(* IEC 61131-3 sources: SmartHomeNew/snapshots/2026-05-07, 56 files *)

(* ---- E_Gateway_Command_Type.dut ---- *)
TYPE E_Gateway_Command_Type :
(
    CMD_NONE := 0,
    CMD_SET_SCENARIO := 1,
    CMD_SET_LIGHT := 2,
    CMD_SET_SOCKET := 3,
    CMD_SET_SECURITY := 4,
    CMD_SET_TEMP := 5,
    CMD_SET_VENT := 6,
    CMD_SET_BLINDS := 7,
    CMD_TELEGRAM_MSG := 8,
    CMD_SYNC_TIME := 9,
    CMD_RESET_ERRORS := 10,
    CMD_SET_CONFIG := 11
) USINT;
END_TYPE

(* ---- E_Outdoor_Mode.dut ---- *)
{attribute 'strict'}
TYPE E_Outdoor_Mode :
(
    OUTDOOR_MODE_AUTO := 0,
    OUTDOOR_MODE_PARTY := 1,
    OUTDOOR_MODE_SECURITY := 2,
    OUTDOOR_MODE_ECONOMY := 3,
    OUTDOOR_MODE_MANUAL := 4
) USINT;
END_TYPE

(* ---- ST_DHW_Status.dut ---- *)
{attribute 'pack_mode' := '1'}
TYPE ST_DHW_Status :
STRUCT
    Temp : REAL;
    Pressure : REAL;
    Heating_Pump_On : BOOL;
    Circ_Pump_On : BOOL;
    Warning : BOOL;
    Error : BOOL;
    Error_ID : WORD;
END_STRUCT
END_TYPE

(* ---- ST_Heating_Runtime_Adaptive_Intelligence.dut ---- *)
TYPE ST_Heating_Runtime_Adaptive_Intelligence :
STRUCT
    // ======================================================
    // Adaptive analytics visibility
    // Passive analytics only.
    // No adaptive authority exists.
    // ======================================================
    Adaptive_Analytics_Visible : BOOL;
    Adaptive_Analytics_Degraded : BOOL;
    Adaptive_Analytics_Attention : BOOL;

    // ======================================================
    // Adaptive supervision observation
    // ======================================================
    Supervision_Confidence_Observation : UINT;
    Confidence_Degradation_Visible : BOOL;

    // ======================================================
    // Adaptive runtime observation
    // ======================================================
    Adaptive_Runtime_Observation : UINT;
    Adaptive_Runtime_Stability_Observation : UINT;

    // ======================================================
    // Adaptive anomaly observation weighting
    // ======================================================
    Runtime_Anomaly_Observation_Weight : UINT;
    Cascade_Anomaly_Observation_Weight : UINT;
    OpenTherm_Anomaly_Observation_Weight : UINT;
    Diagnostics_Anomaly_Observation_Weight : UINT;

    // ======================================================
    // Predictive correlation observation
    // ======================================================
    Predictive_Correlation_Observation : UINT;
    Predictive_Correlation_Visible : BOOL;

    // ======================================================
    // Adaptive integrity observation
    // ======================================================
    Sequencing_Confidence_Observation : UINT;
    Ownership_Confidence_Observation : UINT;
    Synchronization_Confidence_Observation : UINT;

    // ======================================================
    // Adaptive analytics status
    // ======================================================
    Status_Code : UINT;
    Status_Text : STRING(128);
END_STRUCT
END_TYPE

(* ---- ST_Heating_Runtime_Event_Buffer.dut ---- *)
TYPE ST_Heating_Runtime_Event_Buffer :
STRUCT
    // ======================================================
    // Runtime phase events
    // ======================================================
    Events : ARRAY[1..32] OF ST_Heating_Runtime_Phase_Event;

    // ======================================================
    // Runtime buffer state
    // ======================================================
    Write_Index : UINT;
    Read_Index : UINT;
    Event_Count : UINT;
    Overflow : BOOL;

    // ======================================================
    // Runtime integrity
    // ======================================================
    Ordering_Integrity_Valid : BOOL;
    Isolation_Integrity_Valid : BOOL;
    Lifecycle_Integrity_Valid : BOOL;

    // ======================================================
    // Runtime visibility
    // ======================================================
    Diagnostics_Visibility_Valid : BOOL;
    Explainability_Visibility_Valid : BOOL;

    // ======================================================
    // Runtime ownership integrity
    // ======================================================
    OpenTherm_Ownership_Valid : BOOL;
    Cascade_Ownership_Valid : BOOL;
    Safety_Ownership_Valid : BOOL;

    // ======================================================
    // Runtime status
    // ======================================================
    Status_Code : UINT;
    Status_Text : STRING(128);
END_STRUCT
END_TYPE

(* ---- ST_Heating_Runtime_Phase_Event.dut ---- *)
TYPE ST_Heating_Runtime_Phase_Event :
STRUCT
    // ======================================================
    // Runtime phase
    // ======================================================
    Phase : E_Heating_Runtime_Phase;

    // ======================================================
    // Event lifecycle
    // ======================================================
    Event_Active : BOOL;
    Event_Completed : BOOL;
    Event_Failed : BOOL;

    // ======================================================
    // Runtime timing
    // ======================================================
    Start_Time_MS : UDINT;
    End_Time_MS : UDINT;
    Duration_MS : UDINT;

    // ======================================================
    // Runtime integrity
    // ======================================================
    Ordering_Valid : BOOL;
    Isolation_Valid : BOOL;

    // ======================================================
    // Runtime status
    // ======================================================
    Status_Code : UINT;
    Status_Text : STRING(128);

    // ======================================================
    // Diagnostics visibility
    // ======================================================
    Diagnostics_Visible : BOOL;
    Explainability_Visible : BOOL;

    // ======================================================
    // Safety integrity
    // ======================================================
    Safety_Integrity_Valid : BOOL;

    // ======================================================
    // Ownership integrity
    // ======================================================
    OpenTherm_Ownership_Valid : BOOL;
    Cascade_Ownership_Valid : BOOL;
END_STRUCT
END_TYPE

(* ---- ST_Modbus_Response.dut ---- *)
TYPE ST_Modbus_Response :
STRUCT
    Busy : BOOL;
    Done : BOOL;
    Error : BOOL;
    Error_Code : WORD;
    Read_Value : ARRAY[1..32] OF WORD;
    Last_Sequence : UDINT;
    Last_Update_MS : UDINT;
END_STRUCT
END_TYPE

(* ---- ST_OpenTherm_Status.dut ---- *)
TYPE ST_OpenTherm_Status :
STRUCT
    Raw_Heartbeat : UDINT;
    Raw_Ack_Seq : UDINT;
    Raw_Online : BOOL;
    Raw_Error : BOOL;
    Raw_Flame : BOOL;
    Raw_Modulation_x10 : UINT;
    Raw_Boiler_Temp_x10 : INT;
    Raw_Status_Word : WORD;
    Raw_Error_Code : WORD;

    Adapter_Online : BOOL;
    Adapter_Error : BOOL;
    Command_Ack : BOOL;
    Command_Timeout : BOOL;
    Heartbeat_Timeout : BOOL;

    Last_Heartbeat : UDINT;
    Last_Heartbeat_MS : UDINT;

    // Transport freshness telemetry
    Heartbeat_Age_MS : UDINT;
    Command_Age_MS : UDINT;
    Last_Command_Ack_Seq : UDINT;

    Adapter_State : E_OpenTherm_Adapter_State;
    Error_State : E_OpenTherm_Error;
END_STRUCT
END_TYPE

(* ---- ST_Ventilation_Config.dut ---- *)
{attribute 'pack_mode' := '1'}
TYPE ST_Ventilation_Config :
STRUCT
    CO2_Threshold : REAL := 800.0;
    Humidity_Threshold : REAL := 65.0;
    Night_Mode_Start : TOD := TOD#23:00;
    Night_Mode_End : TOD := TOD#07:00;
END_STRUCT
END_TYPE

(* ---- ST_Zone_Adapt_State.dut ---- *)
TYPE ST_Zone_Adapt_State :
STRUCT
    Zone_Weight : REAL;
    Confidence : REAL;
    Activations : UDINT;
    Success_Count : UDINT;
    Failure_Count : UDINT;
    Success_Rate : REAL;
    Avg_Result_Value : REAL;
    Last_Update_MS : UDINT;
END_STRUCT
END_TYPE

(* ---- GVL_BEHAVIOR_ADAPT.gvl ---- *)
VAR_GLOBAL
    // Scenario behavior weights.
    // Scalar fields are the active compile-safe source used by PRG_Scenario_Engine.
    // The structured value is kept as a repository-level model reference, but active code does not depend on direct component access to it.
    G_Behavior_Weight_Comfort : REAL := 1.0;
    G_Behavior_Weight_Night : REAL := 1.0;
    G_Behavior_Weight_Preheat : REAL := 1.0;
    G_Behavior_Weight_VentBoost : REAL := 1.0;
    G_Behavior_Weight_AccessSecure : REAL := 1.0;

    G_Behavior_Weights : ST_Behavior_Weights := (
        W_Comfort := 1.0,
        W_Night := 1.0,
        W_Preheat := 1.0,
        W_VentBoost := 1.0,
        W_AccessSecure := 1.0
    );

    G_Scenario_Stats : ARRAY[0..10] OF ST_Scenario_Stats;
    G_VentBoost_Zone_Adapt : ARRAY[1..GVL_CONSTANTS.C_MAX_ZONES] OF ST_Zone_Adapt_State;

    G_Adapt_Profile : E_Adapt_Profile := ADAPT_PROFILE_BALANCED;

    G_Adapt_Enabled : BOOL := TRUE;
    G_Adapt_Learning_Rate : REAL := 0.05;
    G_Adapt_Update_Threshold : INT := 5;

    G_Adapt_Min_Confidence : REAL := 0.30;
    G_Adapt_Default_Zone_Weight : REAL := 1.0;

    G_Confidence_Learning_Rate : REAL := 0.05;
    G_Decay_Factor : REAL := 0.995;

    G_Prev_Humidity : ARRAY[1..GVL_CONSTANTS.C_MAX_ZONES] OF REAL;
    G_Prev_Valid : ARRAY[1..GVL_CONSTANTS.C_MAX_ZONES] OF BOOL;
END_VAR
// >>> BULK_SYNC_ANCHOR: GVL_BEHAVIOR_ADAPT <<<

(* ---- GVL_CONFIG_BACKUP.gvl ---- *)
{attribute 'qualified_only'}
VAR_GLOBAL
    // Full snapshot of configuration
    G_Backup_FloorHeating_Configs : ARRAY[1..GVL_CONSTANTS.C_MAX_HEATING_CIRCUITS] OF ST_FloorHeating_Circuit_Config;

    G_Backup_Max_Active_Manifolds : INT := 0;
    G_Backup_Max_Thermal_Budget : REAL := 0.0;

    // Integrity flag
    G_Backup_Valid : BOOL := FALSE;
END_VAR

(* ---- GVL_CONSTANTS.gvl ---- *)
{attribute 'qualified_only'}
VAR_GLOBAL CONSTANT
    // Размеры массивов (конфигурация системы)
    C_MAX_ZONES            : INT := 16;
    C_MAX_LIGHTING_ZONES   : INT := 32;
    C_MAX_HEATING_CIRCUITS : INT := 16;
    C_MAX_CLIMATE_ZONES    : INT := 16;
    C_MAX_LIGHT_ZONES      : INT := 32;
    C_MAX_SOCKETS          : INT := 36;
    C_MAX_BLINDS           : INT := 20;
    C_MAX_ALARMS           : INT := 20;
    C_MAX_RULES            : INT := 20;
    C_MAX_MANIFOLDS        : INT := 5;
    C_MAX_BOILERS          : INT := 2;
    C_MAX_SUPPLY_FANS      : INT := 3;
    C_MAX_EXHAUST_FANS     : INT := 5;
    C_MAX_SECURITY_SENSORS : INT := 15;
    C_MAX_FLOOD_SENSORS    : INT := 12;
    C_MAX_DOOR_SENSORS     : INT := 8;
    C_MAX_CO_SENSORS       : INT := 8;
    C_MAX_METHANE_SENSORS  : INT := 2;
    C_PRIMARY_METHANE_SENSOR_INDEX : INT := 1;
    C_PRIMARY_EFFECTIVE_GAS_INDEX : INT := 1;
    C_MAX_VENT_UNITS       : INT := 8;
    C_MAX_SUPPLY_TEMPS     : INT := 2;
    C_MAX_SMOKE_SENSORS    : INT := 6;
    C_MAX_SCENARIOS        : INT := 6;
    C_MAX_OUTDOOR_ZONES    : INT := 4;
    C_MAX_ACCESS_CODES     : INT := 10;
    C_MAX_WET_ZONES        : INT := 4;
    C_MAX_CALIBRATIONS     : INT := 20;
    C_MAX_MODULES          : INT := 10;
    C_MAX_CLEANING_MODES   : INT := 3;
    C_MAX_ALLOWED_IPS      : INT := 5;
    C_MAX_VENT_SUPPLY_MODES: INT := 3;
    C_MAX_SECURITY_PHONES  : INT := 5;
    C_MAX_FLOOD_VALVES     : INT := 3;
    C_MAX_HUMIDITY_SENSORS : INT := 8;
    C_MAX_CO2_SENSORS      : INT := 8;
    C_MAX_CIRCUITS_PER_MANIFOLD : INT := 4;
    C_MAX_TREND_DATA_POINTS: INT := 100;
    C_MAX_HISTORY_RECORDS  : INT := 100;
    C_MAX_DEBUG_LOGS       : INT := 1000;
    C_MAX_GATEWAY_COMMANDS : INT := 10;
    C_MAX_STATE_SNAPSHOTS  : INT := 10;
    C_MAX_BLACKBOX_RECORDS : INT := 100;
    C_MAX_PRESENCE_HISTORY : INT := 1008;
    C_MAX_MODBUS_REGISTERS : INT := 201;
    C_MAX_DEDUPLICATION_HISTORY : INT := 100;
    C_MAX_NVRAM_RECORDS    : INT := 100;
    C_MAX_NVRAM_DATA       : INT := 128;

    C_MAX_WATER_ZONES      : INT := 32;

    C_ANALOG_RAW_MAX       : WORD := 27648;
    C_ANALOG_4MA_RAW       : WORD := 5529;
    C_ANALOG_3_6MA_RAW     : WORD := 4976;
    C_ANALOG_21MA_RAW      : WORD := 29030;
    C_ANALOG_10V_MAX_RAW   : WORD := 30000;

    C_MS_IN_SECOND         : UDINT := 1000;
    C_MS_IN_MINUTE         : UDINT := 60000;
    C_MS_IN_HOUR           : UDINT := 3600000;
    C_MS_IN_DAY            : UDINT := 86400000;

    C_BOILER_CASCADE_MIN_DEMAND : REAL := 25.0;
    C_BOILER_CASCADE_HIGH_DEMAND : REAL := 250.0;
    C_BOILER_SETPOINT_MIN : REAL := 35.0;
    C_BOILER_SETPOINT_MAX : REAL := 55.0;
    C_MIN_HEATING_MANIFOLD_PRESSURE : REAL := 0.8;
END_VAR

(* ---- GVL_GATEWAY.gvl ---- *)
{attribute 'qualified_only'}
VAR_GLOBAL
    G_Gateway_Command : ST_Gateway_Command;
    G_Gateway_Command_Received : BOOL;
    G_Gateway_Send_2FA : BOOL;
    G_Gateway_2FA_Code : STRING(6);
    G_Gateway_Telegram_Msg : STRING(200);
    G_Gateway_Send_Telegram : BOOL;
    G_Gateway_HMI_Status_Message : STRING(200);
    G_Gateway_Ping_OK : BOOL;
    G_Gateway_Data_Ready : BOOL;
    G_Gateway_Modbus_Registers : ARRAY[0..GVL_CONSTANTS.C_MAX_MODBUS_REGISTERS-1] OF WORD;
    // === SHADOW POLICY EXPORT ===
    G_Shadow_Alert_Active : BOOL;
    G_Shadow_Dominant_Channel : STRING(32);
    G_Shadow_Policy_Summary_Text : STRING(160);
    G_Shadow_Recent_Activity_Text : STRING(160);
    G_Shadow_Rate_Summary_Text : STRING(160);
    G_Shadow_Total_Fallback_Count : UDINT;
    G_Shadow_Total_Recovery_Count : UDINT;

END_VAR

(* ---- GVL_Heating_Runtime_Observation.gvl ---- *)
VAR_GLOBAL
    G_Runtime_Observer_Lifecycle_State : E_Runtime_Observer_Lifecycle_State := E_Runtime_Observer_Lifecycle_State.ROS_INACTIVE;
    G_Runtime_Observer_Lifecycle_Code : UINT := 0;
    G_Runtime_Observer_Lifecycle_Text : STRING(128) := 'Heating runtime observer inactive';
    G_Runtime_Observer_Commissioning_Required : BOOL := TRUE;
    G_Runtime_Observer_Commissioning_Active : BOOL := FALSE;
    G_Runtime_Observer_Commissioning_Complete : BOOL := FALSE;
    G_Runtime_Observation : ST_Heating_Runtime_Observation;
    G_Runtime_Observation_Publication_Valid : BOOL := FALSE;
    G_Runtime_Observation_Stabilization_Complete : BOOL := FALSE;
    G_Runtime_Observation_Operational : BOOL := FALSE;
    G_Runtime_Observation_Valid : BOOL := FALSE;
    G_Runtime_Observer_Ready : BOOL := FALSE;
    G_Runtime_Observer_Fault : BOOL := FALSE;
    G_Runtime_Observation_Status_Code : UINT := 0;
    G_Runtime_Observation_Status_Text : STRING(128) := 'Heating runtime observation inactive';
    G_Runtime_Observation_ReadOnly : BOOL := TRUE;
    G_Runtime_Observation_Governance_Locked : BOOL := TRUE;
END_VAR

(* ---- GVL_LIGHTING_OUTPUT.gvl ---- *)
VAR_GLOBAL
    AO_Lighting_Levels : ARRAY[1..GVL_CONSTANTS.C_MAX_LIGHT_ZONES] OF UINT;
    AO_Blinds_Positions : ARRAY[1..GVL_CONSTANTS.C_MAX_BLINDS] OF UINT;
    DO_Sockets : ARRAY[1..GVL_CONSTANTS.C_MAX_SOCKETS] OF BOOL;
END_VAR

(* ---- GVL_STATE.gvl ---- *)
{attribute 'qualified_only'}
VAR_GLOBAL
    G_Floor_Temps : ARRAY[1..GVL_CONSTANTS.C_MAX_HEATING_CIRCUITS] OF REAL;
    G_Room_Temps : ARRAY[1..GVL_CONSTANTS.C_MAX_ZONES] OF REAL;
    G_Last_Valid_Room_Temps : ARRAY[1..GVL_CONSTANTS.C_MAX_ZONES] OF REAL;
    G_Last_Valid_Floor_Temps : ARRAY[1..GVL_CONSTANTS.C_MAX_HEATING_CIRCUITS] OF REAL;
    G_Temp_Sensor_Fault : ARRAY[1..GVL_CONSTANTS.C_MAX_ZONES] OF BOOL;
    G_Floor_Temp_Sensor_Fault : ARRAY[1..GVL_CONSTANTS.C_MAX_HEATING_CIRCUITS] OF BOOL;
    G_Room_Hum : ARRAY[1..GVL_CONSTANTS.C_MAX_ZONES] OF REAL;
    G_Room_CO2 : ARRAY[1..GVL_CONSTANTS.C_MAX_ZONES] OF REAL;
    G_Motion_Sensors : ARRAY[1..GVL_CONSTANTS.C_MAX_LIGHT_ZONES] OF BOOL;
    G_Door_Sensors : ARRAY[1..GVL_CONSTANTS.C_MAX_DOOR_SENSORS] OF BOOL;
    G_Window_Sensors : ARRAY[1..GVL_CONSTANTS.C_MAX_ZONES] OF BOOL;
    G_Water_Sensors : ARRAY[1..GVL_CONSTANTS.C_MAX_FLOOD_SENSORS] OF BOOL;
    G_Smoke_Sensors : ARRAY[1..GVL_CONSTANTS.C_MAX_SMOKE_SENSORS] OF BOOL;
    G_Methane_Sensors : ARRAY[1..GVL_CONSTANTS.C_MAX_METHANE_SENSORS] OF REAL;
    G_CO_Sensors : ARRAY[1..GVL_CONSTANTS.C_MAX_CO_SENSORS] OF REAL;
    G_Manifold_Pressures : ARRAY[1..GVL_CONSTANTS.C_MAX_MANIFOLDS] OF REAL;
    G_Manifold_Currents : ARRAY[1..GVL_CONSTANTS.C_MAX_MANIFOLDS] OF REAL;
    G_Predictive_Pump_Pressure_Drop : ARRAY[1..GVL_CONSTANTS.C_MAX_MANIFOLDS] OF BOOL;
    G_Predictive_Pump_Current_Rise : ARRAY[1..GVL_CONSTANTS.C_MAX_MANIFOLDS] OF BOOL;
    G_Manifold_T_Supply : ARRAY[1..GVL_CONSTANTS.C_MAX_MANIFOLDS] OF REAL;
    G_Manifold_T_Return : ARRAY[1..GVL_CONSTANTS.C_MAX_MANIFOLDS] OF REAL;
    G_Boiler_Flame : ARRAY[1..GVL_CONSTANTS.C_MAX_BOILERS] OF BOOL;
    G_Boiler_Error : ARRAY[1..GVL_CONSTANTS.C_MAX_BOILERS] OF BOOL;
    G_Boiler_OT_Online : ARRAY[1..GVL_CONSTANTS.C_MAX_BOILERS] OF BOOL;
    G_Boiler_OT_Command_Ack : ARRAY[1..GVL_CONSTANTS.C_MAX_BOILERS] OF BOOL;
    G_Boiler_OT_Command_Timeout : ARRAY[1..GVL_CONSTANTS.C_MAX_BOILERS] OF BOOL;
    G_Boiler_OT_Heartbeat_Timeout : ARRAY[1..GVL_CONSTANTS.C_MAX_BOILERS] OF BOOL;
    G_Boiler_OT_Adapter_Error : ARRAY[1..GVL_CONSTANTS.C_MAX_BOILERS] OF BOOL;
    G_Boiler_OT_Heartbeat_Age_MS : ARRAY[1..GVL_CONSTANTS.C_MAX_BOILERS] OF UDINT;
    G_Boiler_OT_Command_Age_MS : ARRAY[1..GVL_CONSTANTS.C_MAX_BOILERS] OF UDINT;
    G_Boiler_OT_Adapter_State : ARRAY[1..GVL_CONSTANTS.C_MAX_BOILERS] OF E_OpenTherm_Adapter_State;
    G_Boiler_OT_Error_State : ARRAY[1..GVL_CONSTANTS.C_MAX_BOILERS] OF E_OpenTherm_Error;
    G_Boiler_OT_Enable : ARRAY[1..GVL_CONSTANTS.C_MAX_BOILERS] OF BOOL;
    G_Boiler_OT_Setpoint : ARRAY[1..GVL_CONSTANTS.C_MAX_BOILERS] OF REAL;

    // Heating cascade semantic aggregate state
    G_Heating_Cascade_Available : BOOL;
    G_Heating_Cascade_Degraded : BOOL;
    G_Heating_Cascade_Partial_Capacity : BOOL;
    G_Heating_Cascade_No_Flame : BOOL;
    G_Heating_Cascade_Transport_Degraded : BOOL;
    G_Heating_Cascade_Ignition_Timeout : BOOL;
    G_Heating_Cascade_Active_Boilers : UINT;
    G_Heating_Cascade_Available_Boilers : UINT;

    G_Physical_Switches : ARRAY[1..GVL_CONSTANTS.C_MAX_LIGHT_ZONES] OF BOOL;
    G_Socket_Switches : ARRAY[1..GVL_CONSTANTS.C_MAX_SOCKETS] OF BOOL;
    G_Outdoor_Temp : REAL;
    G_Supply_Temps : ARRAY[1..GVL_CONSTANTS.C_MAX_SUPPLY_TEMPS] OF REAL;
    G_DHW_Temp : REAL;
    G_DHW_Pressure : REAL;
    G_Zone_Valves : ARRAY[1..GVL_CONSTANTS.C_MAX_HEATING_CIRCUITS] OF BOOL;
    G_Manifold_Pumps : ARRAY[1..GVL_CONSTANTS.C_MAX_MANIFOLDS] OF BOOL;
    G_Manifold_Valves : ARRAY[1..GVL_CONSTANTS.C_MAX_MANIFOLDS] OF REAL;
    G_Manifold_End_Switches : ARRAY[1..GVL_CONSTANTS.C_MAX_MANIFOLDS] OF BOOL;
    G_Supply_Fans : ARRAY[1..GVL_CONSTANTS.C_MAX_SUPPLY_FANS] OF REAL;
    G_Exhaust_Fans : ARRAY[1..GVL_CONSTANTS.C_MAX_EXHAUST_FANS] OF REAL;
    G_Vent_Heater_Power : ARRAY[1..GVL_CONSTANTS.C_MAX_BOILERS] OF REAL;
    G_Lighting_Levels : ARRAY[1..GVL_CONSTANTS.C_MAX_LIGHT_ZONES] OF BYTE;
    G_Blinds_Positions : ARRAY[1..GVL_CONSTANTS.C_MAX_BLINDS] OF BYTE;
    G_Socket_States : ARRAY[1..GVL_CONSTANTS.C_MAX_SOCKETS] OF BOOL;
    G_DHW_Heating_Pump : BOOL;
    G_DHW_Circ_Pump : BOOL;
    G_Backup_Circulation_Pump : BOOL;
    G_Electric_Heater_Enable : BOOL;
    G_Safety_Gas_Alarm : BOOL;
    G_Safety_Leak_Alarm : BOOL;
    G_Safety_Smoke_Alarm : BOOL;
    G_Safety_Emergency_Stop : BOOL;
    G_Safety_Gas_Latched : BOOL;
    G_Safety_Leak_Latched : BOOL;
    G_Safety_Smoke_Latched : BOOL;
    G_Safety_Freeze_Risk : BOOL;
    G_System_Mode : E_System_Operating_Mode := E_System_Operating_Mode.MODE_NORMAL;
    G_System_Mode_Text : STRING(64);
    G_Heating_IO_Fault : BOOL;
    G_Heating_Sensor_Fault : BOOL;
    G_Heating_Subsystem_Degraded : BOOL;
    G_Heating_RootCause : E_Heating_RootCause := E_Heating_RootCause.RC_NONE;
    G_Heating_RootConfidence : REAL;
    G_Heating_Confidence : REAL := 1.0;
    G_Heating_Error_Score : REAL := 0.0;
    G_Heating_Confidence_Reason_Code : INT := 0;
    G_Heating_Confidence_Reason_Text : STRING(128) := 'OK';
    G_DHW_IO_Fault : BOOL;
    G_DHW_Sensor_Fault : BOOL;
    G_DHW_Subsystem_Degraded : BOOL;
    G_Ventilation_IO_Fault : BOOL;
    G_Ventilation_Subsystem_Degraded : BOOL;
    G_Lighting_IO_Fault : BOOL;
    G_Lighting_Subsystem_Degraded : BOOL;
    G_Access_Comm_Fault : BOOL;
    G_Evacuation_Lighting_Active : BOOL;
    G_Evac_Hazard_Zone : ARRAY[1..GVL_CONSTANTS.C_MAX_LIGHT_ZONES] OF BOOL;
    G_Evac_Guidance : ARRAY[1..GVL_CONSTANTS.C_MAX_LIGHT_ZONES] OF INT;

    G_Rule_Actions : ARRAY[1..GVL_CONSTANTS.C_MAX_RULES] OF ST_Rule_Action;
    G_Sim_Lights : ARRAY[1..GVL_CONSTANTS.C_MAX_LIGHT_ZONES] OF BOOL;
    G_Freeze_Hardware_Degraded : BOOL;
    G_Freeze_Hardware_Failed : BOOL;
    G_Water_Zone_Enable : ARRAY[1..GVL_CONSTANTS.C_MAX_WATER_ZONES] OF BOOL;
    G_Water_Zone_Open_FB : ARRAY[1..GVL_CONSTANTS.C_MAX_WATER_ZONES] OF BOOL;
    G_Water_Zone_Close_FB : ARRAY[1..GVL_CONSTANTS.C_MAX_WATER_ZONES] OF BOOL;
    G_Water_Zone_Exercise_Active : ARRAY[1..GVL_CONSTANTS.C_MAX_WATER_ZONES] OF BOOL;
    G_Preheat_Request : BOOL;
    G_Freeze_Request : BOOL;
    G_Target_Temperature : REAL;
END_VAR

(* ---- GVL_STATUS.gvl ---- *)
{attribute 'qualified_only'}
VAR_GLOBAL
    G_System_Time_MS : UDINT;
    G_Last_System_Time_MS : UDINT := 0;
    G_Time_Of_Day_MS : UDINT := 0;
    G_Current_Day : UINT := 1;
    G_Day_Of_Year : UINT := 1;
    G_Current_TOD : TOD;
    G_Current_Scenario : E_SCENARIO_TYPE := E_SCENARIO_TYPE.SCENARIO_NONE;
    G_Previous_Scenario : E_SCENARIO_TYPE := E_SCENARIO_TYPE.SCENARIO_NONE;
    G_Is_Night : BOOL;
    G_PLC_ID : BYTE := 1;
    G_Is_Active_PLC : BOOL;
    G_Other_PLC_Is_Active : BOOL;

    G_Remote_PLC_Last_Seen_MS : UDINT;
    G_Remote_PLC_Alive : BOOL;

    G_Local_PLC_ID : BYTE := 1;
    G_Active_PLC_ID : BYTE := 1;
    G_Remote_PLC_Pulse : BOOL;

    G_Security_Status_Msg : STRING(200);
    G_Gas_Status_Msg : STRING(200);
    G_Flood_Status_Msg : STRING(200);
    G_Vent_Status_Msg : STRING(200);

    G_DHW_Status : ST_DHW_Status;
    G_Manifold_Status : ARRAY[1..GVL_CONSTANTS.C_MAX_MANIFOLDS] OF ST_Manifold_Status;
    G_Boiler_Status : ARRAY[1..GVL_CONSTANTS.C_MAX_BOILERS] OF ST_Boiler_Status;

    G_IO_Modules_Online : ARRAY[1..GVL_CONSTANTS.C_MAX_MODULES] OF BOOL;

    G_Sim_Active : BOOL;
    G_Wet_Zone_Light_Active : BOOL;

    G_System_Mode_Msg : STRING(200);
    G_System_Mode_Cause : STRING(200);
    G_System_Mode_Text : STRING(200);

    G_Evac_Target_Zone_Name : STRING(80);
    G_Evac_Hazard_Zone_Name : STRING(80);

    G_Diagnostics : ST_System_Diagnostics;
    G_Diagnostics_Events : ARRAY[1..50] OF ST_Diagnostic_Event;
    G_Diagnostics_Count : INT := 0;
END_VAR

(* ---- F_Modbus_RTU_CRC16.st ---- *)
FUNCTION F_Modbus_RTU_CRC16 : WORD
VAR_INPUT
    VI_Data : ARRAY[0..255] OF BYTE;
    VI_Length : UINT;
END_VAR

// ======================================================
// LEGACY CRC16 COMPATIBILITY FUNCTION
// ======================================================
// Kept only for backward compatibility.
// Active runtime now uses inline CRC implementations
// inside TX builder, RX parser and SysCom backend.
// ======================================================

F_Modbus_RTU_CRC16 := WORD#16#FFFF;

END_FUNCTION

(* ---- FB_CRC32_Calculator.st ---- *)
FUNCTION_BLOCK FB_CRC32_Calculator
VAR_INPUT
    VI_Enable : BOOL := TRUE;
END_VAR

VAR_OUTPUT
    VO_CRC : DWORD;
END_VAR

VAR
    L_Table : ARRAY[0..255] OF DWORD;
    L_Initialized : BOOL := FALSE;
END_VAR

// Compatibility placeholder.
// Previous METHOD Calculate returned DWORD#0.
// Keep same behaviour without METHOD syntax for this CODESYS project format.
IF VI_Enable THEN
    VO_CRC := DWORD#0;
END_IF;

END_FUNCTION_BLOCK

(* ---- FB_Heating_Circuit_Control.st ---- *)
// ==============================================================================
// Heating circuit control helper
//
// Internal refactoring helper for FB_Heating_System_Manager.
// Owns per-circuit sensor validation, temperature source fallback,
// floor-heating controller call, overheat shutdown, and rule action projection.
// ==============================================================================
FUNCTION_BLOCK FB_Heating_Circuit_Control
VAR_INPUT
    VI_System_Time_MS : UDINT;
    VI_Current_Hour : UINT;
    VI_IsActivePLC : BOOL;
    VI_Config : ST_Heating_Config;
    VI_Tariff : ST_Tariff_Config;
    VI_Scenario_Adjust : REAL;
END_VAR

VAR_IN_OUT
    VI_Zone_Configs : ARRAY[1..GVL_CONSTANTS.C_MAX_HEATING_CIRCUITS] OF ST_FloorHeating_Circuit_Config;
    VI_Floor_Temps : ARRAY[1..GVL_CONSTANTS.C_MAX_HEATING_CIRCUITS] OF REAL;
    VI_Room_Temps : ARRAY[1..16] OF REAL;
    VI_Rule_Actions : ARRAY[1..GVL_CONSTANTS.C_MAX_RULES] OF ST_Rule_Action;
END_VAR

VAR_OUTPUT
    VO_Zone_Valves : ARRAY[1..GVL_CONSTANTS.C_MAX_HEATING_CIRCUITS] OF BOOL;
    VO_Heating_Sensor_Fault : BOOL;
END_VAR

VAR
    L_i : INT;
    L_j : INT;
    L_Climate_Zone_ID : INT;
    L_Zone_Config : ST_FloorHeating_Circuit_Config;
    L_Current_Temp : REAL;
    L_Sensor_Error : BOOL;

    L_Floor_Controllers : ARRAY[1..GVL_CONSTANTS.C_MAX_HEATING_CIRCUITS] OF FB_FloorHeating_Controller;
    L_Overheat_Timer : ARRAY[1..GVL_CONSTANTS.C_MAX_HEATING_CIRCUITS] OF FB_System_Timer;
    fbFloorTempValidator : ARRAY[1..GVL_CONSTANTS.C_MAX_HEATING_CIRCUITS] OF FB_Analog_Validator;
    fbRoomTempValidator : ARRAY[1..16] OF FB_Analog_Validator;
END_VAR

VO_Heating_Sensor_Fault := FALSE;

FOR L_i := 1 TO GVL_CONSTANTS.C_MAX_HEATING_CIRCUITS DO
    fbFloorTempValidator[L_i](
        VI_Value := VI_Floor_Temps[L_i],
        VI_Min_Valid := -40.0,
        VI_Max_Valid := 120.0,
        VI_Fallback_Mode := 0
    );

    L_Climate_Zone_ID := VI_Zone_Configs[L_i].zone;
    IF L_Climate_Zone_ID >= 1 AND L_Climate_Zone_ID <= 16 THEN
        fbRoomTempValidator[L_Climate_Zone_ID](
            VI_Value := VI_Room_Temps[L_Climate_Zone_ID],
            VI_Min_Valid := -40.0,
            VI_Max_Valid := 120.0,
            VI_Fallback_Mode := 0
        );
    END_IF;

    // Floor overheat protection
    L_Overheat_Timer[L_i](
        IN := fbFloorTempValidator[L_i].VO_Value > VI_Config.Overheat_Threshold,
        PT := T#60s,
        VI_System_Time_MS := VI_System_Time_MS
    );

    L_Current_Temp := 0.0;
    L_Sensor_Error := FALSE;

    IF VI_Zone_Configs[L_i].control_type = 1 OR VI_Zone_Configs[L_i].control_type = 2 THEN
        // Primary: room air temperature
        IF (L_Climate_Zone_ID >= 1) AND (L_Climate_Zone_ID <= 16) AND (NOT fbRoomTempValidator[L_Climate_Zone_ID].VO_Error) THEN
            L_Current_Temp := fbRoomTempValidator[L_Climate_Zone_ID].VO_Value;
        ELSIF NOT fbFloorTempValidator[L_i].VO_Error THEN
            L_Current_Temp := fbFloorTempValidator[L_i].VO_Value;
        ELSE
            L_Sensor_Error := TRUE;
        END_IF;
    ELSE
        // Primary: floor temperature
        IF NOT fbFloorTempValidator[L_i].VO_Error THEN
            L_Current_Temp := fbFloorTempValidator[L_i].VO_Value;
        ELSIF (L_Climate_Zone_ID >= 1) AND (L_Climate_Zone_ID <= 16) AND (NOT fbRoomTempValidator[L_Climate_Zone_ID].VO_Error) THEN
            L_Current_Temp := fbRoomTempValidator[L_Climate_Zone_ID].VO_Value;
        ELSE
            L_Sensor_Error := TRUE;
        END_IF;
    END_IF;

    IF L_Sensor_Error THEN
        VO_Heating_Sensor_Fault := TRUE;
        VO_Zone_Valves[L_i] := FALSE;
    ELSE
        L_Zone_Config := VI_Zone_Configs[L_i];
        L_Zone_Config.design_temp := L_Zone_Config.design_temp + VI_Scenario_Adjust;

        L_Floor_Controllers[L_i](
            VI_Current_Temp := L_Current_Temp,
            VI_Config := L_Zone_Config,
            VI_Tariff := VI_Tariff,
            VI_Current_Hour := VI_Current_Hour,
            VI_IsActivePLC := VI_IsActivePLC,
            VI_System_Time_MS := VI_System_Time_MS,
            VO_Valve_Bool => VO_Zone_Valves[L_i]
        );
    END_IF;

    IF L_Overheat_Timer[L_i].Q THEN
        VO_Zone_Valves[L_i] := FALSE;
    END_IF;

    FOR L_j := 1 TO GVL_CONSTANTS.C_MAX_RULES DO
        IF VI_Rule_Actions[L_j].Active AND VI_Rule_Actions[L_j].Target_ID = L_i THEN
            IF VI_Rule_Actions[L_j].Action_Type = E_Rule_Action_Type.ACTION_SET_FLOOR_HEATING THEN
                VO_Zone_Valves[L_i] := (VI_Rule_Actions[L_j].Value > 0.5);
            END_IF;
        END_IF;
    END_FOR;
END_FOR;

// >>> BULK_SYNC_ANCHOR: FB_Heating_Circuit_Control <<<
END_FUNCTION_BLOCK

(* ---- FB_Heating_Diagnostics.st ---- *)
// ==============================================================================
// Heating diagnostics event projection
// Read-only diagnostics layer for service/OOS/freeze hardware events.
// Does NOT own heating control or output decisions.
// ==============================================================================
FUNCTION_BLOCK FB_Heating_Diagnostics
VAR_INPUT
    VI_System_Time_MS : UDINT;
END_VAR
VAR
    fbDiagEventManager : FB_Diagnostics_Event_Manager;
    L_i : INT;
    L_Any_Heating_Device_OOS : BOOL;
    L_Critical_Fault : BOOL;
    L_Device_Text : STRING(200);
    L_Critical_Text : STRING(200);
    L_Event_Text : STRING(200);
    L_Add_Text : STRING(80);
END_VAR

// ======================================================
// DEFAULTS
// ======================================================
L_Any_Heating_Device_OOS := FALSE;
L_Critical_Fault := FALSE;
L_Device_Text := '';
L_Critical_Text := '';
L_Event_Text := '';
L_Add_Text := '';

// ======================================================
// SERVICE / OUT-OF-SERVICE FLAGS
// ======================================================
GVL_STATUS.G_Diagnostics.Backup_Pump_Out_Of_Service :=
    NOT GVL_CONFIG.G_Backup_Circulation_Pump_In_Service;

GVL_STATUS.G_Diagnostics.Electric_Heater_Out_Of_Service :=
    NOT GVL_CONFIG.G_Electric_Heater_In_Service;

IF GVL_STATUS.G_Diagnostics.Backup_Pump_Out_Of_Service THEN
    L_Any_Heating_Device_OOS := TRUE;
    L_Add_Text := 'backup pump out of service';
    L_Device_Text := L_Add_Text;
END_IF;

IF GVL_STATUS.G_Diagnostics.Electric_Heater_Out_Of_Service THEN
    L_Any_Heating_Device_OOS := TRUE;
    L_Add_Text := 'electric heater out of service';
    IF LEN(L_Device_Text) = 0 THEN
        L_Device_Text := L_Add_Text;
    ELSIF (LEN(L_Device_Text) + LEN(L_Add_Text) + 2) < 200 THEN
        L_Device_Text := CONCAT(L_Device_Text, CONCAT('; ', L_Add_Text));
    END_IF;
END_IF;

fbDiagEventManager(
    VI_Code := GVL_CONFIG.ERR_BACKUP_PUMP_OUT_OF_SERVICE,
    VI_Severity := 2,
    VI_Active := GVL_STATUS.G_Diagnostics.Backup_Pump_Out_Of_Service,
    VI_Timestamp := VI_System_Time_MS,
    VI_Source := 400,
    VIO_Events := GVL_STATUS.G_Diagnostics_Events,
    VIO_Count := GVL_STATUS.G_Diagnostics_Count
);

fbDiagEventManager(
    VI_Code := GVL_CONFIG.ERR_ELECTRIC_HEATER_OUT_OF_SERVICE,
    VI_Severity := 2,
    VI_Active := GVL_STATUS.G_Diagnostics.Electric_Heater_Out_Of_Service,
    VI_Timestamp := VI_System_Time_MS,
    VI_Source := 401,
    VIO_Events := GVL_STATUS.G_Diagnostics_Events,
    VIO_Count := GVL_STATUS.G_Diagnostics_Count
);

FOR L_i := 1 TO GVL_CONSTANTS.C_MAX_MANIFOLDS DO

    GVL_STATUS.G_Diagnostics.Manifold_Pump_Out_Of_Service[L_i] :=
        NOT GVL_CONFIG.G_Manifold_Pump_In_Service[L_i];

    IF GVL_STATUS.G_Diagnostics.Manifold_Pump_Out_Of_Service[L_i] THEN
        L_Any_Heating_Device_OOS := TRUE;
        L_Add_Text := CONCAT('manifold pump OOS #', INT_TO_STRING(L_i));

        IF LEN(L_Device_Text) = 0 THEN
            L_Device_Text := L_Add_Text;
        ELSIF (LEN(L_Device_Text) + LEN(L_Add_Text) + 2) < 200 THEN
            L_Device_Text := CONCAT(L_Device_Text, CONCAT('; ', L_Add_Text));
        END_IF;
    END_IF;

    fbDiagEventManager(
        VI_Code := GVL_CONFIG.ERR_MANIFOLD_PUMP_OUT_OF_SERVICE,
        VI_Severity := 2,
        VI_Active := GVL_STATUS.G_Diagnostics.Manifold_Pump_Out_Of_Service[L_i],
        VI_Timestamp := VI_System_Time_MS,
        VI_Source := 410 + L_i,
        VIO_Events := GVL_STATUS.G_Diagnostics_Events,
        VIO_Count := GVL_STATUS.G_Diagnostics_Count
    );

END_FOR;

GVL_STATUS.G_Diagnostics.DHW_Heating_Pump_Out_Of_Service :=
    NOT GVL_CONFIG.G_DHW_Heating_Pump_In_Service;

GVL_STATUS.G_Diagnostics.DHW_Circ_Pump_Out_Of_Service :=
    NOT GVL_CONFIG.G_DHW_Circ_Pump_In_Service;

IF GVL_STATUS.G_Diagnostics.DHW_Heating_Pump_Out_Of_Service THEN
    L_Any_Heating_Device_OOS := TRUE;
    L_Add_Text := 'DHW heating pump out of service';

    IF LEN(L_Device_Text) = 0 THEN
        L_Device_Text := L_Add_Text;
    ELSIF (LEN(L_Device_Text) + LEN(L_Add_Text) + 2) < 200 THEN
        L_Device_Text := CONCAT(L_Device_Text, CONCAT('; ', L_Add_Text));
    END_IF;
END_IF;

IF GVL_STATUS.G_Diagnostics.DHW_Circ_Pump_Out_Of_Service THEN
    L_Any_Heating_Device_OOS := TRUE;
    L_Add_Text := 'DHW circ pump out of service';

    IF LEN(L_Device_Text) = 0 THEN
        L_Device_Text := L_Add_Text;
    ELSIF (LEN(L_Device_Text) + LEN(L_Add_Text) + 2) < 200 THEN
        L_Device_Text := CONCAT(L_Device_Text, CONCAT('; ', L_Add_Text));
    END_IF;
END_IF;

fbDiagEventManager(
    VI_Code := GVL_CONFIG.ERR_DHW_HEATING_PUMP_OUT_OF_SERVICE,
    VI_Severity := 2,
    VI_Active := GVL_STATUS.G_Diagnostics.DHW_Heating_Pump_Out_Of_Service,
    VI_Timestamp := VI_System_Time_MS,
    VI_Source := 420,
    VIO_Events := GVL_STATUS.G_Diagnostics_Events,
    VIO_Count := GVL_STATUS.G_Diagnostics_Count
);

fbDiagEventManager(
    VI_Code := GVL_CONFIG.ERR_DHW_CIRC_PUMP_OUT_OF_SERVICE,
    VI_Severity := 2,
    VI_Active := GVL_STATUS.G_Diagnostics.DHW_Circ_Pump_Out_Of_Service,
    VI_Timestamp := VI_System_Time_MS,
    VI_Source := 421,
    VIO_Events := GVL_STATUS.G_Diagnostics_Events,
    VIO_Count := GVL_STATUS.G_Diagnostics_Count
);

// ======================================================
// FREEZE HARDWARE EVENT PROJECTION
// ======================================================
L_Critical_Fault := GVL_STATE.G_Freeze_Hardware_Failed;

IF L_Critical_Fault THEN
    L_Critical_Text := 'Freeze hardware critical fault';
END_IF;

fbDiagEventManager(
    VI_Code := GVL_CONFIG.ERR_FREEZE_HARDWARE_FAILED,
    VI_Severity := 4,
    VI_Active := L_Critical_Fault,
    VI_Timestamp := VI_System_Time_MS,
    VI_Source := 430,
    VIO_Events := GVL_STATUS.G_Diagnostics_Events,
    VIO_Count := GVL_STATUS.G_Diagnostics_Count
);

GVL_STATUS.G_Diagnostics.Freeze_Hardware_Event_Pending :=
    GVL_STATUS.G_Diagnostics.Freeze_Hardware_Event_Pending OR
    L_Critical_Fault OR
    L_Any_Heating_Device_OOS;

IF L_Critical_Fault AND L_Any_Heating_Device_OOS THEN
    L_Event_Text := CONCAT(L_Critical_Text, '; ');
    IF (LEN(L_Event_Text) + LEN(L_Device_Text)) < 200 THEN
        L_Event_Text := CONCAT(L_Event_Text, L_Device_Text);
    END_IF;
    GVL_STATUS.G_Diagnostics.Freeze_Hardware_Event_Text := L_Event_Text;

ELSIF L_Critical_Fault THEN
    GVL_STATUS.G_Diagnostics.Freeze_Hardware_Event_Text := L_Critical_Text;

ELSIF L_Any_Heating_Device_OOS THEN
    GVL_STATUS.G_Diagnostics.Freeze_Hardware_Event_Text := L_Device_Text;
END_IF;

END_FUNCTION_BLOCK
// >>> BULK_SYNC_ANCHOR: FB_Heating_Diagnostics <<<

(* ---- FB_Heating_Policy_Manager.st ---- *)
FUNCTION_BLOCK FB_Heating_Policy_Manager
VAR_INPUT
    VI_System_Time_MS : UDINT;
    VI_System_Mode : E_System_Operating_Mode;
    VI_RootCause : E_Heating_RootCause;
    VI_RootConfidence : REAL;
    VI_Min_Hold_MS : UDINT;
    VI_Emergency_Stop : BOOL;
    VI_Gas_Safety : BOOL;
    VI_Room_Temp_Avg : REAL;
    VI_Floor_Temp_Avg : REAL;
    VI_Supply_Temp : REAL;
    VI_Return_Temp : REAL;
    VI_Target_Temp : REAL;
    VI_Room_Temps : ARRAY[1..GVL_CONSTANTS.C_MAX_ZONES] OF REAL;
    VI_Floor_Temps : ARRAY[1..GVL_CONSTANTS.C_MAX_ZONES] OF REAL;
END_VAR
VAR_OUTPUT
    VO_Policy_Mode : E_Heating_Policy_Mode;
    VO_Block_Heating : BOOL;
    VO_Target_Adjustment : REAL;
    VO_Priority_Multiplier : REAL;
    VO_Self_Tune_Active : BOOL;
    VO_Self_Tune_Level : INT;
    VO_Feedback_Stable : BOOL;
    VO_Feedback_Improving : BOOL;
    VO_Feedback_Quality : REAL;
END_VAR
VAR
    L_Raw_Mode : E_Heating_Policy_Mode;
    L_Raw_Block : BOOL;
    L_Raw_Target_Adjustment : REAL;
    L_Raw_Priority_Multiplier : REAL;
    L_Held_Mode : E_Heating_Policy_Mode;
    L_Held_Block : BOOL;
    L_Held_Target_Adjustment : REAL;
    L_Held_Priority_Multiplier : REAL;
    L_Last_Accept_MS : UDINT;
    L_Initialized : BOOL;
    L_Effective_Hold_MS : UDINT;
    L_Force_Immediate : BOOL;
    L_Same_Cause_Since : UDINT;
    L_Last_Cause : E_Heating_RootCause;
    L_Self_Level : INT;
    L_Room_Error : REAL;
    L_Supply_Error : REAL;
    L_DeltaT : REAL;
    L_Quality : REAL;
    L_Last_Quality : REAL;
    L_Improving : BOOL;
    L_Stable : BOOL;
    L_Predictive_Initialized : BOOL;
    L_Last_Room_Avg : REAL;
    L_Trend : REAL;
    L_Filtered_Trend : REAL;
    L_Predictive_Adjustment : REAL;
    L_i : INT;
    L_Zone_Error : REAL;
    L_Zone_Quality : REAL;
    L_Last_Zone_Temp : ARRAY[1..GVL_CONSTANTS.C_MAX_ZONES] OF REAL;
    L_Zone_Trend : REAL;
    L_Zone_Filtered_Trend : ARRAY[1..GVL_CONSTANTS.C_MAX_ZONES] OF REAL;
    L_Zone_Desired_Adjustment : REAL;
    L_Zone_Desired_Level : INT;
    L_Zone_Last_Adjust_Accept_MS : ARRAY[1..GVL_CONSTANTS.C_MAX_ZONES] OF UDINT;
    L_Zone_Last_Level_Accept_MS : ARRAY[1..GVL_CONSTANTS.C_MAX_ZONES] OF UDINT;
    L_Zone_Hold_MS : UDINT;
    L_Zone_Inertia : REAL;
    L_Zone_Thermal_Bias : REAL;
    L_Time_To_Heat_MS_REAL : REAL;
END_VAR

L_Zone_Hold_MS := VI_Min_Hold_MS / 2;
IF L_Zone_Hold_MS < 60000 THEN L_Zone_Hold_MS := 60000; END_IF;

IF NOT L_Predictive_Initialized THEN
    L_Last_Room_Avg := VI_Room_Temp_Avg;
    L_Filtered_Trend := 0.0;
    FOR L_i := 1 TO GVL_CONSTANTS.C_MAX_ZONES DO
        L_Last_Zone_Temp[L_i] := VI_Room_Temps[L_i];
        L_Zone_Filtered_Trend[L_i] := 0.0;
        L_Zone_Last_Adjust_Accept_MS[L_i] := VI_System_Time_MS;
        L_Zone_Last_Level_Accept_MS[L_i] := VI_System_Time_MS;
        GVL_HEATING_POLICY.G_Zone_Target_Adjustment[L_i] := 0.0;
        GVL_HEATING_POLICY.G_Zone_Thermal_Response[L_i] := 0.0;
        GVL_HEATING_POLICY.G_Zone_Thermal_Demand[L_i] := 0.0;
        GVL_HEATING_POLICY.G_Zone_Time_To_Heat_MS[L_i] := 0;
        GVL_HEATING_POLICY.G_Zone_Preheat_Needed[L_i] := FALSE;
    END_FOR;
    L_Predictive_Initialized := TRUE;
END_IF;

L_Trend := VI_Room_Temp_Avg - L_Last_Room_Avg;
L_Last_Room_Avg := VI_Room_Temp_Avg;
L_Filtered_Trend := (L_Filtered_Trend * 0.8) + (L_Trend * 0.2);

L_Predictive_Adjustment := 0.0;
IF (L_Filtered_Trend < -0.03) AND (VI_Room_Temp_Avg < (VI_Target_Temp + 0.5)) THEN
    L_Predictive_Adjustment := 1.0;
ELSIF L_Filtered_Trend > 0.03 THEN
    L_Predictive_Adjustment := -0.5;
END_IF;
IF L_Predictive_Adjustment > 1.0 THEN L_Predictive_Adjustment := 1.0; END_IF;
IF L_Predictive_Adjustment < -1.0 THEN L_Predictive_Adjustment := -1.0; END_IF;
GVL_HEATING_POLICY.G_Policy_Predictive_Adjustment := L_Predictive_Adjustment;
GVL_HEATING_POLICY.G_Policy_Predictive_Active := ABS(L_Predictive_Adjustment) > 0.001;

L_Room_Error := VI_Target_Temp - VI_Room_Temp_Avg;
L_Supply_Error := VI_Target_Temp - VI_Supply_Temp;
L_DeltaT := VI_Supply_Temp - VI_Return_Temp;
L_Quality := 0.0;
IF L_Room_Error > 1.0 THEN L_Quality := L_Quality + 2.0; END_IF;
IF L_Supply_Error > 1.0 THEN L_Quality := L_Quality + 1.0; END_IF;
IF L_DeltaT < 3.0 THEN L_Quality := L_Quality + 1.0; END_IF;
L_Improving := L_Quality < L_Last_Quality;
L_Stable := L_Quality = 0.0;

FOR L_i := 1 TO GVL_CONSTANTS.C_MAX_ZONES DO
    L_Zone_Error := VI_Target_Temp - VI_Room_Temps[L_i];
    L_Zone_Quality := 0.0;
    IF L_Zone_Error > 1.0 THEN L_Zone_Quality := L_Zone_Quality + 2.0; END_IF;
    IF VI_Floor_Temps[L_i] < (VI_Target_Temp - 2.0) THEN L_Zone_Quality := L_Zone_Quality + 1.0; END_IF;

    L_Zone_Trend := VI_Room_Temps[L_i] - L_Last_Zone_Temp[L_i];
    L_Last_Zone_Temp[L_i] := VI_Room_Temps[L_i];
    L_Zone_Filtered_Trend[L_i] := (L_Zone_Filtered_Trend[L_i] * 0.8) + (L_Zone_Trend * 0.2);

    L_Zone_Inertia := GVL_HEATING_POLICY.G_Zone_Thermal_Inertia[L_i];
    IF L_Zone_Inertia < 0.2 THEN L_Zone_Inertia := 1.0; END_IF;
    IF L_Zone_Inertia > 3.0 THEN L_Zone_Inertia := 3.0; END_IF;

    GVL_HEATING_POLICY.G_Zone_Thermal_Response[L_i] := L_Zone_Filtered_Trend[L_i] / L_Zone_Inertia;
    GVL_HEATING_POLICY.G_Zone_Thermal_Demand[L_i] := L_Zone_Error * L_Zone_Inertia;

    IF (L_Zone_Error > 0.0) AND (GVL_HEATING_POLICY.G_Zone_Thermal_Response[L_i] > 0.001) THEN
        L_Time_To_Heat_MS_REAL := (L_Zone_Error / GVL_HEATING_POLICY.G_Zone_Thermal_Response[L_i]) * 60000.0;
        IF L_Time_To_Heat_MS_REAL > 7200000.0 THEN
            GVL_HEATING_POLICY.G_Zone_Time_To_Heat_MS[L_i] := 7200000;
        ELSIF L_Time_To_Heat_MS_REAL < 0.0 THEN
            GVL_HEATING_POLICY.G_Zone_Time_To_Heat_MS[L_i] := 0;
        ELSE
            GVL_HEATING_POLICY.G_Zone_Time_To_Heat_MS[L_i] := REAL_TO_UDINT(L_Time_To_Heat_MS_REAL);
        END_IF;
    ELSE
        GVL_HEATING_POLICY.G_Zone_Time_To_Heat_MS[L_i] := 0;
    END_IF;

    GVL_HEATING_POLICY.G_Zone_Preheat_Needed[L_i] := (GVL_HEATING_POLICY.G_Zone_Time_To_Heat_MS[L_i] > 1800000) AND (L_Zone_Error > 0.5);

    L_Zone_Thermal_Bias := 0.0;
    IF GVL_HEATING_POLICY.G_Zone_Thermal_Demand[L_i] > 2.0 THEN
        L_Zone_Thermal_Bias := 0.5;
    ELSIF GVL_HEATING_POLICY.G_Zone_Thermal_Demand[L_i] > 1.0 THEN
        L_Zone_Thermal_Bias := 0.25;
    ELSIF GVL_HEATING_POLICY.G_Zone_Thermal_Demand[L_i] < -1.0 THEN
        L_Zone_Thermal_Bias := -0.4;
    END_IF;

    IF GVL_HEATING_POLICY.G_Zone_Preheat_Needed[L_i] THEN
        L_Zone_Thermal_Bias := L_Zone_Thermal_Bias + 0.4;
    END_IF;

    L_Zone_Desired_Adjustment := L_Zone_Thermal_Bias;
    IF (L_Zone_Filtered_Trend[L_i] < -0.03) AND (VI_Room_Temps[L_i] < (VI_Target_Temp + 0.5)) THEN
        L_Zone_Desired_Adjustment := L_Zone_Desired_Adjustment + 0.8;
    ELSIF L_Zone_Filtered_Trend[L_i] > 0.03 THEN
        L_Zone_Desired_Adjustment := L_Zone_Desired_Adjustment - 0.3;
    END_IF;
    IF L_Zone_Desired_Adjustment > 1.0 THEN L_Zone_Desired_Adjustment := 1.0; END_IF;
    IF L_Zone_Desired_Adjustment < -1.0 THEN L_Zone_Desired_Adjustment := -1.0; END_IF;

    IF ABS(L_Zone_Desired_Adjustment - GVL_HEATING_POLICY.G_Zone_Target_Adjustment[L_i]) > 0.001 THEN
        IF (VI_System_Time_MS - L_Zone_Last_Adjust_Accept_MS[L_i]) >= L_Zone_Hold_MS THEN
            GVL_HEATING_POLICY.G_Zone_Target_Adjustment[L_i] := L_Zone_Desired_Adjustment;
            L_Zone_Last_Adjust_Accept_MS[L_i] := VI_System_Time_MS;
        END_IF;
    END_IF;

    GVL_HEATING_POLICY.G_Zone_Improving[L_i] := (L_Zone_Quality < GVL_HEATING_POLICY.G_Zone_Quality[L_i]);
    GVL_HEATING_POLICY.G_Zone_Stable[L_i] := (L_Zone_Quality = 0.0);

    L_Zone_Desired_Level := GVL_HEATING_POLICY.G_Zone_Self_Level[L_i];
    IF GVL_HEATING_POLICY.G_Zone_Stable[L_i] THEN
        L_Zone_Desired_Level := 0;
    ELSIF GVL_HEATING_POLICY.G_Zone_Improving[L_i] THEN
        L_Zone_Desired_Level := GVL_HEATING_POLICY.G_Zone_Self_Level[L_i] - 1;
    ELSIF L_Zone_Quality >= 3.0 THEN
        L_Zone_Desired_Level := GVL_HEATING_POLICY.G_Zone_Self_Level[L_i] + 1;
    END_IF;
    IF L_Zone_Desired_Level > 2 THEN L_Zone_Desired_Level := 2; END_IF;
    IF L_Zone_Desired_Level < 0 THEN L_Zone_Desired_Level := 0; END_IF;
    IF L_Zone_Desired_Level <> GVL_HEATING_POLICY.G_Zone_Self_Level[L_i] THEN
        IF (VI_System_Time_MS - L_Zone_Last_Level_Accept_MS[L_i]) >= L_Zone_Hold_MS THEN
            GVL_HEATING_POLICY.G_Zone_Self_Level[L_i] := L_Zone_Desired_Level;
            L_Zone_Last_Level_Accept_MS[L_i] := VI_System_Time_MS;
        END_IF;
    END_IF;

    GVL_HEATING_POLICY.G_Zone_Quality[L_i] := L_Zone_Quality;
END_FOR;

IF VI_RootCause <> L_Last_Cause THEN
    L_Same_Cause_Since := VI_System_Time_MS;
    L_Self_Level := 0;
END_IF;
L_Last_Cause := VI_RootCause;

IF L_Stable THEN
    L_Self_Level := 0;
ELSIF L_Improving THEN
    L_Self_Level := L_Self_Level - 1;
ELSIF (VI_System_Time_MS - L_Same_Cause_Since) > (VI_Min_Hold_MS * 2) AND (VI_RootConfidence > 0.8) AND (L_Quality >= 3.0) THEN
    L_Self_Level := L_Self_Level + 1;
END_IF;
IF L_Self_Level > 2 THEN L_Self_Level := 2; END_IF;
IF L_Self_Level < 0 THEN L_Self_Level := 0; END_IF;

L_Raw_Mode := E_Heating_Policy_Mode.HPM_NORMAL;
L_Raw_Block := FALSE;
L_Raw_Target_Adjustment := L_Predictive_Adjustment;
L_Raw_Priority_Multiplier := 1.0;
L_Force_Immediate := FALSE;

IF VI_Emergency_Stop OR VI_Gas_Safety THEN
    L_Raw_Mode := E_Heating_Policy_Mode.HPM_SAFETY_BLOCK;
    L_Raw_Block := TRUE;
    L_Raw_Target_Adjustment := 0.0;
    L_Raw_Priority_Multiplier := 1.0;
    L_Force_Immediate := TRUE;
ELSIF VI_RootCause = E_Heating_RootCause.RC_IO_OFFLINE THEN
    L_Raw_Mode := E_Heating_Policy_Mode.HPM_DEGRADED;
    L_Raw_Block := TRUE;
    L_Raw_Target_Adjustment := 0.0;
    L_Raw_Priority_Multiplier := 1.0;
    L_Force_Immediate := TRUE;
ELSIF VI_RootConfidence >= 0.6 THEN
    CASE VI_RootCause OF
        E_Heating_RootCause.RC_NO_HEAT_TRANSFER:
            L_Raw_Mode := E_Heating_Policy_Mode.HPM_DEGRADED;
            L_Raw_Target_Adjustment := L_Raw_Target_Adjustment + 3.0 + TO_REAL(L_Self_Level);
        E_Heating_RootCause.RC_PUMP_FAILURE:
            L_Raw_Mode := E_Heating_Policy_Mode.HPM_FAULT_ISOLATION;
            L_Raw_Priority_Multiplier := 0.5 - (0.1 * TO_REAL(L_Self_Level));
        E_Heating_RootCause.RC_VALVES_CLOSED:
            L_Raw_Mode := E_Heating_Policy_Mode.HPM_FAULT_ISOLATION;
            L_Raw_Target_Adjustment := L_Raw_Target_Adjustment - 2.0;
        E_Heating_RootCause.RC_NO_FLAME,
        E_Heating_RootCause.RC_BOILER_ERROR:
            L_Raw_Mode := E_Heating_Policy_Mode.HPM_DEGRADED;
            L_Raw_Priority_Multiplier := 0.7;
        ELSE
            IF VI_System_Mode = E_System_Operating_Mode.MODE_DEGRADED THEN L_Raw_Mode := E_Heating_Policy_Mode.HPM_DEGRADED; END_IF;
    END_CASE;
ELSE
    IF VI_System_Mode = E_System_Operating_Mode.MODE_DEGRADED THEN L_Raw_Mode := E_Heating_Policy_Mode.HPM_DEGRADED; END_IF;
END_IF;

IF L_Raw_Target_Adjustment > 5.0 THEN L_Raw_Target_Adjustment := 5.0; END_IF;
IF L_Raw_Target_Adjustment < -3.0 THEN L_Raw_Target_Adjustment := -3.0; END_IF;
IF L_Raw_Priority_Multiplier < 0.3 THEN L_Raw_Priority_Multiplier := 0.3; END_IF;
IF L_Raw_Priority_Multiplier > 1.0 THEN L_Raw_Priority_Multiplier := 1.0; END_IF;

L_Effective_Hold_MS := VI_Min_Hold_MS;
IF VI_RootConfidence >= 0.9 THEN L_Effective_Hold_MS := VI_Min_Hold_MS / 2; END_IF;

IF NOT L_Initialized THEN
    L_Held_Mode := L_Raw_Mode;
    L_Held_Block := L_Raw_Block;
    L_Held_Target_Adjustment := L_Raw_Target_Adjustment;
    L_Held_Priority_Multiplier := L_Raw_Priority_Multiplier;
    L_Last_Accept_MS := VI_System_Time_MS;
    L_Initialized := TRUE;
ELSIF L_Force_Immediate THEN
    L_Held_Mode := L_Raw_Mode;
    L_Held_Block := L_Raw_Block;
    L_Held_Target_Adjustment := L_Raw_Target_Adjustment;
    L_Held_Priority_Multiplier := L_Raw_Priority_Multiplier;
    L_Last_Accept_MS := VI_System_Time_MS;
ELSIF (L_Raw_Mode <> L_Held_Mode) OR (ABS(L_Raw_Target_Adjustment - L_Held_Target_Adjustment) > 0.001) OR (ABS(L_Raw_Priority_Multiplier - L_Held_Priority_Multiplier) > 0.001) OR (L_Raw_Block <> L_Held_Block) THEN
    IF (VI_System_Time_MS - L_Last_Accept_MS) >= L_Effective_Hold_MS THEN
        L_Held_Mode := L_Raw_Mode;
        L_Held_Block := L_Raw_Block;
        L_Held_Target_Adjustment := L_Raw_Target_Adjustment;
        L_Held_Priority_Multiplier := L_Raw_Priority_Multiplier;
        L_Last_Accept_MS := VI_System_Time_MS;
    END_IF;
END_IF;

VO_Policy_Mode := L_Held_Mode;
VO_Block_Heating := L_Held_Block;
VO_Target_Adjustment := L_Held_Target_Adjustment;
VO_Priority_Multiplier := L_Held_Priority_Multiplier;
VO_Self_Tune_Active := (L_Self_Level > 0);
VO_Self_Tune_Level := L_Self_Level;
VO_Feedback_Stable := L_Stable;
VO_Feedback_Improving := L_Improving;
VO_Feedback_Quality := L_Quality;
L_Last_Quality := L_Quality;

END_FUNCTION_BLOCK

(* ---- FB_Heating_Runtime_Adaptive_Risk_Scorer.st ---- *)
// ==============================================================================
// Heating runtime adaptive risk scorer
// Read-only adaptive supervision scoring layer.
// ==============================================================================
FUNCTION_BLOCK FB_Heating_Runtime_Adaptive_Risk_Scorer
VAR_INPUT
    VI_Enable : BOOL;
    VI_Runtime_Degraded : BOOL;
    VI_Runtime_Critical : BOOL;
END_VAR
VAR_OUTPUT
    VO_Adaptive_Runtime_Risk : UINT;
    VO_Adaptive_Runtime_Stability : UINT;

    VO_Status_Code : UINT;
    VO_Status_Text : STRING(128);
END_VAR

VO_Adaptive_Runtime_Risk := 0;
VO_Adaptive_Runtime_Stability := 100;

VO_Status_Code := 0;
VO_Status_Text := 'Heating adaptive risk scorer disabled';

IF NOT VI_Enable THEN
    RETURN;
END_IF;

IF VI_Runtime_Critical THEN
    VO_Adaptive_Runtime_Risk := 100;
    VO_Adaptive_Runtime_Stability := 0;

    VO_Status_Code := 900;
    VO_Status_Text := 'Heating runtime adaptive risk critical';

ELSIF VI_Runtime_Degraded THEN
    VO_Adaptive_Runtime_Risk := 60;
    VO_Adaptive_Runtime_Stability := 40;

    VO_Status_Code := 200;
    VO_Status_Text := 'Heating runtime adaptive degradation';

ELSE
    VO_Adaptive_Runtime_Risk := 5;
    VO_Adaptive_Runtime_Stability := 95;

    VO_Status_Code := 1;
    VO_Status_Text := 'Heating runtime adaptive supervision nominal';
END_IF;

END_FUNCTION_BLOCK
// >>> BULK_SYNC_ANCHOR: FB_Heating_Runtime_Adaptive_Risk_Scorer <<<

(* ---- FB_Heating_Runtime_Anomaly_Correlator.st ---- *)
// ==============================================================================
// Heating runtime anomaly correlator
// Read-only runtime anomaly correlation layer.
// ==============================================================================
FUNCTION_BLOCK FB_Heating_Runtime_Anomaly_Correlator
VAR_INPUT
    VI_Enable : BOOL;
    VI_Runtime_Jitter : BOOL;
    VI_Runtime_Latency : BOOL;
    VI_Runtime_Degraded : BOOL;
    VI_Sequencing_Valid : BOOL;
    VI_Ownership_Valid : BOOL;
    VI_Synchronization_Valid : BOOL;
END_VAR
VAR_OUTPUT
    VO_Anomaly : ST_Heating_Runtime_Anomaly;
END_VAR

VO_Anomaly.Anomaly_Active := FALSE;
VO_Anomaly.Anomaly_Acknowledged := FALSE;
VO_Anomaly.Anomaly_Cleared := FALSE;

VO_Anomaly.Status_Code := 0;
VO_Anomaly.Status_Text := 'Heating runtime anomaly correlator disabled';

IF NOT VI_Enable THEN
    RETURN;
END_IF;

VO_Anomaly.Runtime_Jitter_Detected := VI_Runtime_Jitter;
VO_Anomaly.Runtime_Latency_Detected := VI_Runtime_Latency;
VO_Anomaly.Runtime_Degraded := VI_Runtime_Degraded;

VO_Anomaly.Sequencing_Invalid := NOT VI_Sequencing_Valid;
VO_Anomaly.Ownership_Invalid := NOT VI_Ownership_Valid;
VO_Anomaly.Synchronization_Invalid := NOT VI_Synchronization_Valid;

VO_Anomaly.Anomaly_Active :=
    VI_Runtime_Jitter OR
    VI_Runtime_Latency OR
    VI_Runtime_Degraded OR
    NOT VI_Sequencing_Valid OR
    NOT VI_Ownership_Valid OR
    NOT VI_Synchronization_Valid;

IF VO_Anomaly.Anomaly_Active THEN
    VO_Anomaly.Status_Code := 100;
    VO_Anomaly.Status_Text := 'Heating runtime anomaly detected';
ELSE
    VO_Anomaly.Status_Code := 1;
    VO_Anomaly.Status_Text := 'Heating runtime nominal';
END_IF;

END_FUNCTION_BLOCK
// >>> BULK_SYNC_ANCHOR: FB_Heating_Runtime_Anomaly_Correlator <<<

(* ---- FB_Heating_Runtime_Anomaly_Severity_Classifier.st ---- *)
// ==============================================================================
// Heating runtime anomaly severity classifier
// Read-only runtime anomaly severity classification layer.
// ==============================================================================
FUNCTION_BLOCK FB_Heating_Runtime_Anomaly_Severity_Classifier
VAR_INPUT
    VI_Enable : BOOL;
    VI_Anomaly : ST_Heating_Runtime_Anomaly;
END_VAR
VAR_OUTPUT
    VO_Severity_Level : UINT;
    VO_Critical_Anomaly : BOOL;

    VO_Status_Code : UINT;
    VO_Status_Text : STRING(128);
END_VAR

VO_Severity_Level := 0;
VO_Critical_Anomaly := FALSE;

VO_Status_Code := 0;
VO_Status_Text := 'Heating runtime anomaly severity classifier disabled';

IF NOT VI_Enable THEN
    RETURN;
END_IF;

IF VI_Anomaly.Ownership_Invalid OR
   VI_Anomaly.Sequencing_Invalid OR
   VI_Anomaly.Synchronization_Invalid THEN

    VO_Severity_Level := 100;
    VO_Critical_Anomaly := TRUE;

    VO_Status_Code := 900;
    VO_Status_Text := 'Heating runtime anomaly critical';

ELSIF VI_Anomaly.Runtime_Degraded OR
       VI_Anomaly.Cascade_Degraded OR
       VI_Anomaly.OpenTherm_Transport_Degraded THEN

    VO_Severity_Level := 50;

    VO_Status_Code := 200;
    VO_Status_Text := 'Heating runtime anomaly degraded';

ELSIF VI_Anomaly.Anomaly_Active THEN

    VO_Severity_Level := 10;

    VO_Status_Code := 100;
    VO_Status_Text := 'Heating runtime anomaly detected';

ELSE
    VO_Severity_Level := 0;

    VO_Status_Code := 1;
    VO_Status_Text := 'Heating runtime anomaly nominal';
END_IF;

END_FUNCTION_BLOCK
// >>> BULK_SYNC_ANCHOR: FB_Heating_Runtime_Anomaly_Severity_Classifier <<<

(* ---- FB_Heating_Runtime_Confidence_Decay_Analyzer.st ---- *)
// ==============================================================================
// Heating runtime confidence decay analyzer
// Read-only predictive confidence decay layer.
// ==============================================================================
FUNCTION_BLOCK FB_Heating_Runtime_Confidence_Decay_Analyzer
VAR_INPUT
    VI_Enable : BOOL;
    VI_Confidence : UINT;
END_VAR
VAR_OUTPUT
    VO_Decay_Detected : BOOL;
    VO_Decay_Score : UINT;

    VO_Status_Code : UINT;
    VO_Status_Text : STRING(128);
END_VAR

VO_Decay_Detected := FALSE;
VO_Decay_Score := 0;

VO_Status_Code := 0;
VO_Status_Text := 'Heating confidence decay analyzer disabled';

IF NOT VI_Enable THEN
    RETURN;
END_IF;

IF VI_Confidence < 40 THEN
    VO_Decay_Detected := TRUE;
    VO_Decay_Score := 90;

    VO_Status_Code := 900;
    VO_Status_Text := 'Heating supervision confidence critical decay';

ELSIF VI_Confidence < 70 THEN
    VO_Decay_Detected := TRUE;
    VO_Decay_Score := 50;

    VO_Status_Code := 200;
    VO_Status_Text := 'Heating supervision confidence degraded';

ELSE
    VO_Decay_Score := 5;

    VO_Status_Code := 1;
    VO_Status_Text := 'Heating supervision confidence nominal';
END_IF;

END_FUNCTION_BLOCK
// >>> BULK_SYNC_ANCHOR: FB_Heating_Runtime_Confidence_Decay_Analyzer <<<

(* ---- FB_Heating_Runtime_Contract_Validator.st ---- *)
// ==============================================================================
// Heating runtime contract validator
// Read-only orchestration validation layer.
// DOES NOT own runtime.
// DOES NOT own heating logic.
// DOES NOT own diagnostics.
// DOES NOT own OpenTherm transport.
// ==============================================================================
FUNCTION_BLOCK FB_Heating_Runtime_Contract_Validator
VAR_INPUT
    VI_Context : ST_Heating_Runtime_Context;
END_VAR
VAR_OUTPUT
    VO_Contract_Valid : BOOL;
    VO_Runtime_Ordering_Valid : BOOL;
    VO_Runtime_Isolation_Valid : BOOL;
    VO_Runtime_Status_Code : UINT;
    VO_Runtime_Status_Text : STRING(128);
END_VAR
VAR
    L_Ordering_Valid : BOOL;
    L_Isolation_Valid : BOOL;
    L_Contract_Valid : BOOL;
END_VAR

// ======================================================
// DEFAULTS
// ======================================================
VO_Contract_Valid := FALSE;
VO_Runtime_Ordering_Valid := FALSE;
VO_Runtime_Isolation_Valid := FALSE;
VO_Runtime_Status_Code := 0;
VO_Runtime_Status_Text := 'Heating runtime contract validator idle';

L_Ordering_Valid := TRUE;
L_Isolation_Valid := TRUE;
L_Contract_Valid := TRUE;

// ======================================================
// RUNTIME ORDERING VALIDATION
// ======================================================
IF NOT VI_Context.DHW_Before_Heating_Valid THEN
    L_Ordering_Valid := FALSE;
END_IF;

IF NOT VI_Context.State_Publication_Before_Diagnostics_Valid THEN
    L_Ordering_Valid := FALSE;
END_IF;

IF NOT VI_Context.Output_Projection_Last_Valid THEN
    L_Ordering_Valid := FALSE;
END_IF;

// ======================================================
// EXECUTION CONSISTENCY VALIDATION
// ======================================================
IF VI_Context.Heating_Executed AND NOT VI_Context.DHW_Executed THEN
    L_Ordering_Valid := FALSE;
END_IF;

IF VI_Context.Diagnostics_Executed AND NOT VI_Context.State_Publication_Executed THEN
    L_Ordering_Valid := FALSE;
END_IF;

IF VI_Context.Output_Projection_Executed AND NOT VI_Context.Diagnostics_Executed THEN
    L_Ordering_Valid := FALSE;
END_IF;

// ======================================================
// OWNERSHIP / ISOLATION VALIDATION
// ======================================================
IF NOT VI_Context.Diagnostics_Isolation_Valid THEN
    L_Isolation_Valid := FALSE;
END_IF;

IF NOT VI_Context.Explainability_Isolation_Valid THEN
    L_Isolation_Valid := FALSE;
END_IF;

IF NOT VI_Context.Safety_Isolation_Valid THEN
    L_Isolation_Valid := FALSE;
END_IF;

IF NOT VI_Context.OpenTherm_Ownership_Valid THEN
    L_Isolation_Valid := FALSE;
END_IF;

IF NOT VI_Context.Cascade_Ownership_Valid THEN
    L_Isolation_Valid := FALSE;
END_IF;

// ======================================================
// FINAL CONTRACT VALIDATION
// ======================================================
L_Contract_Valid :=
    L_Ordering_Valid AND
    L_Isolation_Valid AND
    NOT VI_Context.Runtime_Fault;

VO_Runtime_Ordering_Valid := L_Ordering_Valid;
VO_Runtime_Isolation_Valid := L_Isolation_Valid;
VO_Contract_Valid := L_Contract_Valid;

// ======================================================
// STATUS
// ======================================================
IF NOT L_Ordering_Valid THEN
    VO_Runtime_Status_Code := 100;
    VO_Runtime_Status_Text := 'Heating runtime ordering validation failed';

ELSIF NOT L_Isolation_Valid THEN
    VO_Runtime_Status_Code := 200;
    VO_Runtime_Status_Text := 'Heating runtime ownership isolation failed';

ELSIF VI_Context.Runtime_Fault THEN
    VO_Runtime_Status_Code := 300;
    VO_Runtime_Status_Text := 'Heating runtime fault active';

ELSE
    VO_Runtime_Status_Code := 1;
    VO_Runtime_Status_Text := 'Heating runtime contract valid';
END_IF;

END_FUNCTION_BLOCK
// >>> BULK_SYNC_ANCHOR: FB_Heating_Runtime_Contract_Validator <<<

(* ---- FB_Heating_Runtime_Degradation_Timeline_Rebuilder.st ---- *)
// ==============================================================================
// Heating runtime degradation timeline rebuilder
// Read-only runtime degradation reconstruction layer.
// ==============================================================================
FUNCTION_BLOCK FB_Heating_Runtime_Degradation_Timeline_Rebuilder
VAR_INPUT
    VI_Enable : BOOL;
    VI_Event : ST_Heating_Runtime_Blackbox_Event;
END_VAR
VAR_IN_OUT
    VIO_Timeline : ST_Heating_Runtime_Blackbox_Timeline;
END_VAR
VAR
    L_Index : UINT;
END_VAR

IF NOT VI_Enable THEN
    RETURN;
END_IF;

// ======================================================
// SAFE INDEX NORMALIZATION
// ======================================================
IF (VIO_Timeline.Write_Index < 1) OR
   (VIO_Timeline.Write_Index >= 256) THEN

    L_Index := 1;

    IF VIO_Timeline.Write_Index >= 256 THEN
        VIO_Timeline.Timeline_Overflow := TRUE;
    END_IF;

ELSE
    L_Index := VIO_Timeline.Write_Index + 1;
END_IF;

// ======================================================
// EVENT STORAGE
// ======================================================
VIO_Timeline.Events[L_Index] := VI_Event;
VIO_Timeline.Write_Index := L_Index;

IF VIO_Timeline.Event_Count < 256 THEN
    VIO_Timeline.Event_Count :=
        VIO_Timeline.Event_Count + 1;
END_IF;

// ======================================================
// PASSIVE FORENSIC VISIBILITY
// ======================================================
VIO_Timeline.Reconstruction_Visible := TRUE;
VIO_Timeline.Forensic_Timeline_Visible :=
    VI_Event.Event_Active;

VIO_Timeline.Root_Cause_Reconstructed :=
    VI_Event.Root_Cause_Candidate;

// ======================================================
// TIMELINE INTEGRITY
// ======================================================
VIO_Timeline.Sequencing_Valid :=
    NOT VI_Event.Sequencing_Invalid;

VIO_Timeline.Ownership_Valid :=
    NOT VI_Event.Ownership_Invalid;

VIO_Timeline.Synchronization_Valid :=
    NOT VI_Event.Synchronization_Invalid;

// ======================================================
// STATUS
// ======================================================
IF VI_Event.Root_Cause_Candidate THEN
    VIO_Timeline.Status_Code := 900;
    VIO_Timeline.Status_Text := 'Heating runtime degradation reconstructed';
ELSE
    VIO_Timeline.Status_Code := 1;
    VIO_Timeline.Status_Text := 'Heating runtime forensic timeline nominal';
END_IF;

END_FUNCTION_BLOCK
// >>> BULK_SYNC_ANCHOR: FB_Heating_Runtime_Degradation_Timeline_Rebuilder <<<

(* ---- FB_Heating_Runtime_Health_Observer.st ---- *)
// ==============================================================================
// Heating runtime health observer
// Read-only orchestration health aggregation layer.
// DOES NOT own runtime.
// DOES NOT own heating logic.
// DOES NOT own diagnostics.
// DOES NOT own OpenTherm transport.
// DOES NOT own migration.
// ==============================================================================
FUNCTION_BLOCK FB_Heating_Runtime_Health_Observer
VAR_INPUT
    VI_Enable : BOOL;
    VI_Context : ST_Heating_Runtime_Context;
    VI_Bridge : ST_Heating_Runtime_Integration_Bridge;

    VI_Synchronized : BOOL;
    VI_Phase_Synchronized : BOOL;
    VI_Ownership_Synchronized : BOOL;
    VI_Sequencing_Synchronized : BOOL;
END_VAR
VAR_OUTPUT
    VO_Runtime_Healthy : BOOL;
    VO_Runtime_Degraded : BOOL;
    VO_Runtime_Critical : BOOL;

    VO_Sequencing_Healthy : BOOL;
    VO_Ownership_Healthy : BOOL;
    VO_Synchronization_Healthy : BOOL;

    VO_Status_Code : UINT;
    VO_Status_Text : STRING(128);
END_VAR
VAR
    L_Healthy : BOOL;
    L_Degraded : BOOL;
    L_Critical : BOOL;
END_VAR

// ======================================================
// DEFAULTS
// ======================================================
VO_Runtime_Healthy := FALSE;
VO_Runtime_Degraded := FALSE;
VO_Runtime_Critical := FALSE;

VO_Sequencing_Healthy := FALSE;
VO_Ownership_Healthy := FALSE;
VO_Synchronization_Healthy := FALSE;

VO_Status_Code := 0;
VO_Status_Text := 'Heating runtime health observer disabled';

L_Healthy := TRUE;
L_Degraded := FALSE;
L_Critical := FALSE;

IF NOT VI_Enable THEN
    RETURN;
END_IF;

// ======================================================
// SEQUENCING HEALTH
// ======================================================
VO_Sequencing_Healthy :=
    VI_Bridge.DHW_Before_Heating_Valid AND
    VI_Bridge.Diagnostics_After_Publication_Valid AND
    VI_Bridge.Output_Projection_Last_Valid AND
    VI_Sequencing_Synchronized;

IF NOT VO_Sequencing_Healthy THEN
    L_Healthy := FALSE;
    L_Degraded := TRUE;
END_IF;

// ======================================================
// OWNERSHIP HEALTH
// ======================================================
VO_Ownership_Healthy :=
    VI_Bridge.Runtime_Ownership_Valid AND
    VI_Bridge.Diagnostics_Ownership_Valid AND
    VI_Bridge.Explainability_Ownership_Valid AND
    VI_Bridge.OpenTherm_Ownership_Valid AND
    VI_Bridge.Cascade_Ownership_Valid AND
    VI_Bridge.Safety_Ownership_Valid AND
    VI_Ownership_Synchronized;

IF NOT VO_Ownership_Healthy THEN
    L_Healthy := FALSE;
    L_Critical := TRUE;
END_IF;

// ======================================================
// SYNCHRONIZATION HEALTH
// ======================================================
VO_Synchronization_Healthy :=
    VI_Synchronized AND
    VI_Phase_Synchronized;

IF NOT VO_Synchronization_Healthy THEN
    L_Healthy := FALSE;
    L_Degraded := TRUE;
END_IF;

// ======================================================
// CONTEXT HEALTH
// ======================================================
IF VI_Context.Runtime_Fault THEN
    L_Healthy := FALSE;
    L_Critical := TRUE;
END_IF;

IF NOT VI_Bridge.Runtime_Migration_Allowed THEN
    L_Healthy := FALSE;
    L_Degraded := TRUE;
END_IF;

// ======================================================
// FINAL HEALTH
// ======================================================
VO_Runtime_Healthy :=
    L_Healthy AND
    NOT L_Degraded AND
    NOT L_Critical;

VO_Runtime_Degraded :=
    L_Degraded AND
    NOT L_Critical;

VO_Runtime_Critical := L_Critical;

// ======================================================
// STATUS
// ======================================================
IF L_Critical THEN
    VO_Status_Code := 900;
    VO_Status_Text := 'Heating runtime orchestration critical';

ELSIF L_Degraded THEN
    VO_Status_Code := 200;
    VO_Status_Text := 'Heating runtime orchestration degraded';

ELSE
    VO_Status_Code := 1;
    VO_Status_Text := 'Heating runtime orchestration healthy';
END_IF;

END_FUNCTION_BLOCK
// >>> BULK_SYNC_ANCHOR: FB_Heating_Runtime_Health_Observer <<<

(* ---- FB_Heating_Runtime_Integration_Bridge_Manager.st ---- *)
// ==============================================================================
// Heating runtime integration bridge manager
// Read-only orchestration integration layer.
// DOES NOT own runtime.
// DOES NOT own heating logic.
// DOES NOT own diagnostics.
// DOES NOT own OpenTherm transport.
// DOES NOT connect orchestration to live runtime yet.
// ==============================================================================
FUNCTION_BLOCK FB_Heating_Runtime_Integration_Bridge_Manager
VAR_INPUT
    VI_Enable : BOOL;
    VI_Runtime_Context : ST_Heating_Runtime_Context;
    VI_Contract_Valid : BOOL;
END_VAR
VAR_OUTPUT
    VO_Bridge : ST_Heating_Runtime_Integration_Bridge;

    VO_Bridge_Ready : BOOL;
    VO_Bridge_Fault : BOOL;
    VO_Bridge_Status_Code : UINT;
    VO_Bridge_Status_Text : STRING(128);
END_VAR

// ======================================================
// DEFAULTS
// ======================================================
VO_Bridge.Shell_Ready := FALSE;
VO_Bridge.Shell_Fault := FALSE;
VO_Bridge.Shell_Contract_Valid := FALSE;

VO_Bridge.Allow_DHW_Integration := FALSE;
VO_Bridge.Allow_Heating_Integration := FALSE;
VO_Bridge.Allow_Diagnostics_Integration := FALSE;
VO_Bridge.Allow_Output_Projection_Integration := FALSE;

VO_Bridge.Runtime_Ownership_Valid := TRUE;
VO_Bridge.Diagnostics_Ownership_Valid := TRUE;
VO_Bridge.Explainability_Ownership_Valid := TRUE;
VO_Bridge.OpenTherm_Ownership_Valid := TRUE;
VO_Bridge.Cascade_Ownership_Valid := TRUE;
VO_Bridge.Safety_Ownership_Valid := TRUE;

VO_Bridge.DHW_Before_Heating_Valid := TRUE;
VO_Bridge.Diagnostics_After_Publication_Valid := TRUE;
VO_Bridge.Output_Projection_Last_Valid := TRUE;

// ======================================================
// GOVERNANCE LOCK
// Observation-only bridge.
// No migration authority exists here.
// ======================================================
VO_Bridge.Governance_Locked := TRUE;
VO_Bridge.Runtime_Attachment_Allowed := FALSE;
VO_Bridge.Runtime_Attachment_Active := FALSE;

VO_Bridge.Integration_Status_Code := 0;
VO_Bridge.Integration_Status_Text := 'Heating runtime bridge disabled';

VO_Bridge.Diagnostics_Visible := TRUE;
VO_Bridge.Explainability_Visible := TRUE;

VO_Bridge.Current_Phase := E_Heating_Runtime_Phase.HRP_DISABLED;
VO_Bridge.Runtime_Synchronized := FALSE;

VO_Bridge_Ready := FALSE;
VO_Bridge_Fault := FALSE;
VO_Bridge_Status_Code := 0;
VO_Bridge_Status_Text := 'Heating runtime bridge disabled';

IF NOT VI_Enable THEN
    RETURN;
END_IF;

// ======================================================
// SHELL STATE
// ======================================================
VO_Bridge.Shell_Ready := VI_Runtime_Context.Runtime_Ready;
VO_Bridge.Shell_Fault := VI_Runtime_Context.Runtime_Fault;
VO_Bridge.Shell_Contract_Valid := VI_Contract_Valid;

// ======================================================
// OWNERSHIP INTEGRITY
// ======================================================
VO_Bridge.Runtime_Ownership_Valid := TRUE;

VO_Bridge.Diagnostics_Ownership_Valid :=
    VI_Runtime_Context.Diagnostics_Isolation_Valid;

VO_Bridge.Explainability_Ownership_Valid :=
    VI_Runtime_Context.Explainability_Isolation_Valid;

VO_Bridge.OpenTherm_Ownership_Valid :=
    VI_Runtime_Context.OpenTherm_Ownership_Valid;

VO_Bridge.Cascade_Ownership_Valid :=
    VI_Runtime_Context.Cascade_Ownership_Valid;

VO_Bridge.Safety_Ownership_Valid :=
    VI_Runtime_Context.Safety_Isolation_Valid;

// ======================================================
// SEQUENCING INTEGRITY
// ======================================================
VO_Bridge.DHW_Before_Heating_Valid :=
    VI_Runtime_Context.DHW_Before_Heating_Valid;

VO_Bridge.Diagnostics_After_Publication_Valid :=
    VI_Runtime_Context.State_Publication_Before_Diagnostics_Valid;

VO_Bridge.Output_Projection_Last_Valid :=
    VI_Runtime_Context.Output_Projection_Last_Valid;

// ======================================================
// OBSERVATION-ONLY INTEGRATION READINESS
// ======================================================
VO_Bridge.Allow_DHW_Integration :=
    VO_Bridge.DHW_Before_Heating_Valid;

VO_Bridge.Allow_Heating_Integration :=
    VO_Bridge.Runtime_Ownership_Valid AND
    VO_Bridge.Cascade_Ownership_Valid;

VO_Bridge.Allow_Diagnostics_Integration :=
    VO_Bridge.Diagnostics_Ownership_Valid AND
    VO_Bridge.Explainability_Ownership_Valid;

VO_Bridge.Allow_Output_Projection_Integration :=
    VO_Bridge.Output_Projection_Last_Valid;

// ======================================================
// GOVERNANCE POLICY
// Runtime attachment remains externally governed.
// Supervision cannot authorize runtime migration.
// ======================================================
VO_Bridge.Governance_Locked := TRUE;
VO_Bridge.Runtime_Attachment_Allowed := FALSE;
VO_Bridge.Runtime_Attachment_Active := FALSE;

// ======================================================
// PHASE SYNCHRONIZATION
// ======================================================
VO_Bridge.Current_Phase := VI_Runtime_Context.Current_Phase;
VO_Bridge.Runtime_Synchronized := VI_Contract_Valid;

// ======================================================
// STATUS
// ======================================================
IF NOT VI_Contract_Valid THEN
    VO_Bridge.Integration_Status_Code := 100;
    VO_Bridge.Integration_Status_Text := 'Heating runtime contract invalid';

ELSIF VI_Runtime_Context.Runtime_Fault THEN
    VO_Bridge.Integration_Status_Code := 200;
    VO_Bridge.Integration_Status_Text := 'Heating runtime fault active';

ELSIF NOT VO_Bridge.Allow_Heating_Integration THEN
    VO_Bridge.Integration_Status_Code := 300;
    VO_Bridge.Integration_Status_Text := 'Heating observation integration blocked';

ELSE
    VO_Bridge.Integration_Status_Code := 1;
    VO_Bridge.Integration_Status_Text := 'Heating observation bridge ready';
END_IF;

// ======================================================
// OUTPUT STATUS
// ======================================================
VO_Bridge_Ready :=
    VO_Bridge.Allow_Heating_Integration;

VO_Bridge_Fault :=
    NOT VI_Contract_Valid OR
    VI_Runtime_Context.Runtime_Fault;

VO_Bridge_Status_Code :=
    VO_Bridge.Integration_Status_Code;

VO_Bridge_Status_Text :=
    VO_Bridge.Integration_Status_Text;

END_FUNCTION_BLOCK
// >>> BULK_SYNC_ANCHOR: FB_Heating_Runtime_Integration_Bridge_Manager <<<

(* ---- FB_Heating_Runtime_Intelligence_Consistency_Analyzer.st ---- *)
// ==============================================================================
// Heating runtime intelligence consistency analyzer
// Read-only meta-supervision consistency layer.
// ==============================================================================
FUNCTION_BLOCK FB_Heating_Runtime_Intelligence_Consistency_Analyzer
VAR_INPUT
    VI_Enable : BOOL;
    VI_Integrity_Valid : BOOL;
    VI_Drift_Detected : BOOL;
    VI_Decay_Detected : BOOL;
END_VAR
VAR_OUTPUT
    VO_Consistency_Valid : BOOL;
    VO_Consistency_Score : UINT;

    VO_Status_Code : UINT;
    VO_Status_Text : STRING(128);
END_VAR

// ======================================================
// DETERMINISTIC DEFAULTS
// ======================================================
VO_Consistency_Valid := FALSE;
VO_Consistency_Score := 0;

VO_Status_Code := 0;
VO_Status_Text := 'Heating intelligence consistency analyzer disabled';

IF NOT VI_Enable THEN
    RETURN;
END_IF;

// ======================================================
// CONSISTENCY ANALYSIS
// ======================================================
VO_Consistency_Valid :=
    VI_Integrity_Valid AND
    NOT VI_Drift_Detected AND
    NOT VI_Decay_Detected;

IF VO_Consistency_Valid THEN
    VO_Consistency_Score := 95;

    VO_Status_Code := 1;
    VO_Status_Text := 'Heating intelligence consistency nominal';

ELSIF VI_Integrity_Valid THEN
    VO_Consistency_Score := 60;

    VO_Status_Code := 200;
    VO_Status_Text := 'Heating intelligence consistency degraded';

ELSE
    VO_Consistency_Score := 10;

    VO_Status_Code := 900;
    VO_Status_Text := 'Heating intelligence consistency invalid';
END_IF;

END_FUNCTION_BLOCK
// >>> BULK_SYNC_ANCHOR: FB_Heating_Runtime_Intelligence_Consistency_Analyzer <<<

(* ---- FB_Heating_Runtime_Jitter_Detector.st ---- *)
// ==============================================================================
// Heating runtime jitter detector
// Read-only deterministic runtime jitter detector.
// ==============================================================================
FUNCTION_BLOCK FB_Heating_Runtime_Jitter_Detector
VAR_INPUT
    VI_Enable : BOOL;
    VI_Frame_Duration_MS : UDINT;
END_VAR
VAR_OUTPUT
    VO_Jitter_Detected : BOOL;
    VO_Status_Code : UINT;
    VO_Status_Text : STRING(128);
END_VAR

VO_Jitter_Detected := FALSE;
VO_Status_Code := 0;
VO_Status_Text := 'Heating runtime jitter detector disabled';

IF NOT VI_Enable THEN
    RETURN;
END_IF;

IF VI_Frame_Duration_MS > 250 THEN
    VO_Jitter_Detected := TRUE;
    VO_Status_Code := 200;
    VO_Status_Text := 'Heating runtime jitter detected';
ELSE
    VO_Status_Code := 1;
    VO_Status_Text := 'Heating runtime jitter nominal';
END_IF;

END_FUNCTION_BLOCK
// >>> BULK_SYNC_ANCHOR: FB_Heating_Runtime_Jitter_Detector <<<

(* ---- FB_Heating_Runtime_Observation_Aggregator.st ---- *)
// ==============================================================================
// Heating runtime observation aggregator
// Read-only orchestration observation aggregation layer.
// ==============================================================================
FUNCTION_BLOCK FB_Heating_Runtime_Observation_Aggregator
VAR_INPUT
    VI_Enable : BOOL;
    VI_Observation : ST_Heating_Runtime_Observation;
    VI_Observation_Valid : BOOL;
END_VAR
VAR_OUTPUT
    VO_Runtime_Healthy : BOOL;
    VO_Runtime_Degraded : BOOL;
    VO_Runtime_Critical : BOOL;

    VO_Status_Code : UINT;
    VO_Status_Text : STRING(128);
END_VAR

VO_Runtime_Healthy := FALSE;
VO_Runtime_Degraded := FALSE;
VO_Runtime_Critical := FALSE;

VO_Status_Code := 0;
VO_Status_Text := 'Heating runtime observation aggregator disabled';

IF NOT VI_Enable THEN
    RETURN;
END_IF;

IF NOT VI_Observation_Valid THEN
    VO_Runtime_Critical := TRUE;
    VO_Status_Code := 900;
    VO_Status_Text := 'Heating runtime observation invalid';

ELSIF VI_Observation.Runtime_Fault THEN
    VO_Runtime_Critical := TRUE;
    VO_Status_Code := 901;
    VO_Status_Text := 'Heating runtime fault observed';

ELSIF VI_Observation.Cascade_Degraded OR
      VI_Observation.OpenTherm_Transport_Degraded THEN

    VO_Runtime_Degraded := TRUE;
    VO_Status_Code := 200;
    VO_Status_Text := 'Heating runtime degraded';

ELSE
    VO_Runtime_Healthy := TRUE;
    VO_Status_Code := 1;
    VO_Status_Text := 'Heating runtime healthy';
END_IF;

END_FUNCTION_BLOCK
// >>> BULK_SYNC_ANCHOR: FB_Heating_Runtime_Observation_Aggregator <<<

(* ---- FB_Heating_Runtime_Observation_Validator.st ---- *)
// ==============================================================================
// Heating runtime observation validator
// Read-only observation validation layer.
// ==============================================================================
FUNCTION_BLOCK FB_Heating_Runtime_Observation_Validator
VAR_INPUT
    VI_Enable : BOOL;
    VI_Observation : ST_Heating_Runtime_Observation;
END_VAR
VAR_OUTPUT
    VO_Observation_Valid : BOOL;
    VO_Status_Code : UINT;
    VO_Status_Text : STRING(128);
END_VAR

VO_Observation_Valid := FALSE;
VO_Status_Code := 0;
VO_Status_Text := 'Heating runtime observation validator disabled';

IF NOT VI_Enable THEN
    RETURN;
END_IF;

VO_Observation_Valid :=
    VI_Observation.Runtime_Ownership_Valid AND
    VI_Observation.Diagnostics_Ownership_Valid AND
    VI_Observation.OpenTherm_Ownership_Valid AND
    VI_Observation.Cascade_Ownership_Valid AND
    VI_Observation.Safety_Ownership_Valid AND
    VI_Observation.DHW_Before_Heating_Observed AND
    VI_Observation.Diagnostics_After_Publication_Observed AND
    VI_Observation.Output_Projection_Last_Observed;

IF VO_Observation_Valid THEN
    VO_Status_Code := 1;
    VO_Status_Text := 'Heating runtime observation valid';
ELSE
    VO_Status_Code := 100;
    VO_Status_Text := 'Heating runtime observation invalid';
END_IF;

END_FUNCTION_BLOCK
// >>> BULK_SYNC_ANCHOR: FB_Heating_Runtime_Observation_Validator <<<

(* ---- FB_Heating_Runtime_Phase_Sequencing_Validator.st ---- *)
// ==============================================================================
// Heating runtime phase sequencing validator
// Read-only deterministic sequencing validator.
// ==============================================================================
FUNCTION_BLOCK FB_Heating_Runtime_Phase_Sequencing_Validator
VAR_INPUT
    VI_Enable : BOOL;
    VI_Transition : ST_Heating_Runtime_Phase_Transition;
END_VAR
VAR_OUTPUT
    VO_Sequencing_Valid : BOOL;
    VO_Status_Code : UINT;
    VO_Status_Text : STRING(128);
END_VAR

VO_Sequencing_Valid := FALSE;
VO_Status_Code := 0;
VO_Status_Text := 'Heating runtime sequencing validator disabled';

IF NOT VI_Enable THEN
    RETURN;
END_IF;

VO_Sequencing_Valid :=
    VI_Transition.Sequencing_Valid AND
    VI_Transition.Ownership_Valid AND
    VI_Transition.Synchronization_Valid AND
    NOT VI_Transition.Transition_Failed;

IF VO_Sequencing_Valid THEN
    VO_Status_Code := 1;
    VO_Status_Text := 'Heating runtime sequencing valid';
ELSE
    VO_Status_Code := 100;
    VO_Status_Text := 'Heating runtime sequencing invalid';
END_IF;

END_FUNCTION_BLOCK
// >>> BULK_SYNC_ANCHOR: FB_Heating_Runtime_Phase_Sequencing_Validator <<<

(* ---- FB_Heating_Runtime_Phase_Telemetry_Aggregator.st ---- *)
// ==============================================================================
// Heating runtime phase telemetry aggregator
// Read-only deterministic orchestration telemetry layer.
// ==============================================================================
FUNCTION_BLOCK FB_Heating_Runtime_Phase_Telemetry_Aggregator
VAR_INPUT
    VI_Enable : BOOL;
    VI_Transition : ST_Heating_Runtime_Phase_Transition;
    VI_Sequencing_Valid : BOOL;
END_VAR
VAR_OUTPUT
    VO_Phase_Healthy : BOOL;
    VO_Phase_Degraded : BOOL;
    VO_Phase_Critical : BOOL;

    VO_Status_Code : UINT;
    VO_Status_Text : STRING(128);
END_VAR

VO_Phase_Healthy := FALSE;
VO_Phase_Degraded := FALSE;
VO_Phase_Critical := FALSE;

VO_Status_Code := 0;
VO_Status_Text := 'Heating runtime phase telemetry disabled';

IF NOT VI_Enable THEN
    RETURN;
END_IF;

IF NOT VI_Sequencing_Valid THEN
    VO_Phase_Critical := TRUE;
    VO_Status_Code := 900;
    VO_Status_Text := 'Heating runtime sequencing critical';

ELSIF VI_Transition.Transition_Failed THEN
    VO_Phase_Critical := TRUE;
    VO_Status_Code := 901;
    VO_Status_Text := 'Heating runtime phase transition failed';

ELSIF VI_Transition.Transition_Duration_MS > 5000 THEN
    VO_Phase_Degraded := TRUE;
    VO_Status_Code := 200;
    VO_Status_Text := 'Heating runtime phase transition degraded';

ELSE
    VO_Phase_Healthy := TRUE;
    VO_Status_Code := 1;
    VO_Status_Text := 'Heating runtime phase telemetry healthy';
END_IF;

END_FUNCTION_BLOCK
// >>> BULK_SYNC_ANCHOR: FB_Heating_Runtime_Phase_Telemetry_Aggregator <<<

(* ---- FB_Heating_Runtime_Supervision_Integrity_Validator.st ---- *)
// ==============================================================================
// Heating runtime supervision integrity validator
// Read-only meta-supervision integrity layer.
// ==============================================================================
FUNCTION_BLOCK FB_Heating_Runtime_Supervision_Integrity_Validator
VAR_INPUT
    VI_Enable : BOOL;
    VI_Confidence : UINT;
    VI_Correlation_Score : UINT;
END_VAR
VAR_OUTPUT
    VO_Integrity_Valid : BOOL;
    VO_Integrity_Score : UINT;

    VO_Status_Code : UINT;
    VO_Status_Text : STRING(128);
END_VAR

VO_Integrity_Valid := FALSE;
VO_Integrity_Score := 0;

VO_Status_Code := 0;
VO_Status_Text := 'Heating supervision integrity validator disabled';

IF NOT VI_Enable THEN
    RETURN;
END_IF;

VO_Integrity_Score :=
    (VI_Confidence + VI_Correlation_Score) / 2;

VO_Integrity_Valid :=
    (VO_Integrity_Score >= 60);

IF NOT VO_Integrity_Valid THEN
    VO_Status_Code := 900;
    VO_Status_Text := 'Heating supervision integrity invalid';

ELSIF VO_Integrity_Score < 80 THEN
    VO_Status_Code := 200;
    VO_Status_Text := 'Heating supervision integrity degraded';

ELSE
    VO_Status_Code := 1;
    VO_Status_Text := 'Heating supervision integrity nominal';
END_IF;

END_FUNCTION_BLOCK
// >>> BULK_SYNC_ANCHOR: FB_Heating_Runtime_Supervision_Integrity_Validator <<<

(* ---- FB_HMI_Interface.st ---- *)
FUNCTION_BLOCK FB_HMI_Interface
VAR_INPUT
    VI_Severity   : E_System_Severity;
    VI_RootCause  : E_System_Root_Cause;
    VI_Status_Msg : STRING(200);
END_VAR

VAR_OUTPUT
    VO_HMI_Status_Text : STRING(200);
    VO_HMI_State_Code  : INT;
END_VAR

VO_HMI_Status_Text := VI_Status_Msg;

CASE VI_Severity OF
    E_System_Severity.SEV_NORMAL:
        VO_HMI_State_Code := 0;
    E_System_Severity.SEV_WARNING:
        VO_HMI_State_Code := 1;
    E_System_Severity.SEV_DEGRADED:
        VO_HMI_State_Code := 2;
    E_System_Severity.SEV_CRITICAL:
        VO_HMI_State_Code := 3;
ELSE
        // No fallback required
END_CASE;
// >>> BULK_SYNC_ANCHOR: FB_HMI_Interface <<<
END_FUNCTION_BLOCK

(* ---- FB_Modbus_RTU_RX_Parser.st ---- *)
FUNCTION_BLOCK FB_Modbus_RTU_RX_Parser
VAR_INPUT
    VI_Frame : ST_Modbus_RTU_Frame;
    VI_Expected_Slave_ID : BYTE;
    VI_Expected_Function : E_Modbus_Function;
END_VAR

VAR_OUTPUT
    VO_Valid : BOOL;
    VO_Error : BOOL;
    VO_Error_Code : WORD;
    VO_Exception_Response : BOOL;
    VO_Register_Count : UINT;
    VO_Register_Value : ARRAY[1..32] OF WORD;
END_VAR

VAR
    L_CRC_Calc : WORD;
    L_CRC_Frame : WORD;
    L_Function_Byte : BYTE;
    L_Expected_Function : BYTE;
    L_Byte_Count : UINT;
    L_i : UINT;
    L_j : INT;
    L_Data_Index : UINT;
END_VAR

// ======================================================
// MODBUS RTU RX FRAME PARSER
// ======================================================

VO_Valid := FALSE;
VO_Error := FALSE;
VO_Error_Code := 0;
VO_Exception_Response := FALSE;
VO_Register_Count := 0;

FOR L_i := 1 TO 32 DO
    VO_Register_Value[L_i] := 0;
END_FOR;

IF NOT VI_Frame.Valid THEN
    VO_Error := TRUE;
    VO_Error_Code := 16#0201;
    RETURN;
END_IF;

IF VI_Frame.Length < 5 THEN
    VO_Error := TRUE;
    VO_Error_Code := 16#0202;
    RETURN;
END_IF;

CASE VI_Expected_Function OF
    MB_FC03_READ_HOLDING_REGISTERS:
        L_Expected_Function := 3;
    MB_FC04_READ_INPUT_REGISTERS:
        L_Expected_Function := 4;
    MB_FC06_WRITE_SINGLE_REGISTER:
        L_Expected_Function := 6;
    MB_FC16_WRITE_MULTIPLE_REGISTERS:
        L_Expected_Function := 16;
ELSE
    VO_Error := TRUE;
    VO_Error_Code := 16#0203;
    RETURN;
END_CASE;

// ======================================================
// CRC VALIDATION
// ======================================================
L_CRC_Frame :=
    BYTE_TO_WORD(VI_Frame.Data[VI_Frame.Length - 2]) OR
    SHL(BYTE_TO_WORD(VI_Frame.Data[VI_Frame.Length - 1]), 8);

L_CRC_Calc := 16#FFFF;

FOR L_i := 0 TO (VI_Frame.Length - UINT#3) DO

    L_CRC_Calc := L_CRC_Calc XOR BYTE_TO_WORD(VI_Frame.Data[L_i]);

    FOR L_j := 0 TO 7 DO
        IF (L_CRC_Calc AND 16#0001) <> 0 THEN
            L_CRC_Calc := SHR(L_CRC_Calc, 1);
            L_CRC_Calc := L_CRC_Calc XOR 16#A001;
        ELSE
            L_CRC_Calc := SHR(L_CRC_Calc, 1);
        END_IF;
    END_FOR;

END_FOR;

IF L_CRC_Calc <> L_CRC_Frame THEN
    VO_Error := TRUE;
    VO_Error_Code := 16#0204;
    RETURN;
END_IF;

IF VI_Frame.Data[0] <> VI_Expected_Slave_ID THEN
    VO_Error := TRUE;
    VO_Error_Code := 16#0205;
    RETURN;
END_IF;

L_Function_Byte := VI_Frame.Data[1];

IF L_Function_Byte = (L_Expected_Function OR 16#80) THEN
    VO_Exception_Response := TRUE;
    VO_Error := TRUE;
    VO_Error_Code := 16#0206;
    RETURN;
END_IF;

IF L_Function_Byte <> L_Expected_Function THEN
    VO_Error := TRUE;
    VO_Error_Code := 16#0207;
    RETURN;
END_IF;

CASE VI_Expected_Function OF

    MB_FC03_READ_HOLDING_REGISTERS,
    MB_FC04_READ_INPUT_REGISTERS:

        L_Byte_Count := VI_Frame.Data[2];

        IF (L_Byte_Count = 0) OR ((L_Byte_Count MOD 2) <> 0) THEN
            VO_Error := TRUE;
            VO_Error_Code := 16#0208;
            RETURN;
        END_IF;

        VO_Register_Count := L_Byte_Count / 2;

        IF VO_Register_Count > 32 THEN
            VO_Error := TRUE;
            VO_Error_Code := 16#0209;
            RETURN;
        END_IF;

        L_Data_Index := 3;

        FOR L_i := 1 TO VO_Register_Count DO

            VO_Register_Value[L_i] :=
                SHL(BYTE_TO_WORD(VI_Frame.Data[L_Data_Index]), 8) OR
                BYTE_TO_WORD(VI_Frame.Data[L_Data_Index + 1]);

            L_Data_Index := L_Data_Index + 2;

        END_FOR;

    MB_FC06_WRITE_SINGLE_REGISTER,
    MB_FC16_WRITE_MULTIPLE_REGISTERS:

        VO_Register_Count := 0;

ELSE
    VO_Error := TRUE;
    VO_Error_Code := 16#020A;
    RETURN;
END_CASE;

VO_Valid := TRUE;

END_FUNCTION_BLOCK
